      ;ENDFOLD
      ;FOLD -- ServoGun SZ1 oeffnen -- ;%{SE}%MKUKATPVW %CVW_COM %VCOMMENT %P 2:-- ServoGun SZ1 oeffnen --, 3: VW_COMMENT
      ;ENDFOLD
      ;FOLD A3511 = AUS ;%{SE}%MKUKATPVW %CVW_SPS %VBOASG %P 2:A3511 = AUS, 3: BOASG
         $OUT[3511] = FALSE
      ;ENDFOLD
      ;FOLD A3512 = EIN ;%{SE}%MKUKATPVW %CVW_SPS %VBOASG %P 2:A3512 = EIN, 3: BOASG
         $OUT[3512] = TRUE
      ;ENDFOLD
      ;FOLD -- RSK Fehlerausgabe Kraftaufbau -- ;%{SE}%MKUKATPVW %CVW_COM %VCOMMENT %P 2:-- RSK Fehlerausgabe Kraftaufbau --, 3: VW_COMMENT
      ;ENDFOLD
      ;FOLD F325 = AUS ;%{SE}%MKUKATPVW %CVW_SPS %VBOASG %P 2:F325 = AUS, 3: BOASG
         $FLAG[325] = FALSE
      ;ENDFOLD
      ;FOLD -- RSK Fehlerausgabe -- ;%{SE}%MKUKATPVW %CVW_COM %VCOMMENT %P 2:-- RSK Fehlerausgabe --, 3: VW_COMMENT
      ;ENDFOLD
      ;FOLD F327 = AUS ;%{SE}%MKUKATPVW %CVW_SPS %VBOASG %P 2:F327 = AUS, 3: BOASG
         $FLAG[327] = FALSE
      ;ENDFOLD
      ;FOLD -- RSK Fehlerausgabe -- ;%{SE}%MKUKATPVW %CVW_COM %VCOMMENT %P 2:-- RSK Fehlerausgabe --, 3: VW_COMMENT
      ;ENDFOLD
      ;FOLD F329 = AUS ;%{SE}%MKUKATPVW %CVW_SPS %VBOASG %P 2:F329 = AUS, 3: BOASG
         $FLAG[329] = FALSE
      ;ENDFOLD
      ;FOLD Schritt 234 = A3894 & A3506 & A3505 & !A3507 & A4039 ;%{SE}%MKUKATPVW %CVW_SPS %VST_CON %P 2:Schritt 234 = A3894 & A3506 & A3505 & !A3507 & A4039, 3: ST_CON
         IF $OUT[3894] AND $OUT[3506] AND $OUT[3505] AND NOT $OUT[3507] AND $OUT[4039] THEN
            PREV_STEP[9] = APP_INT_STEP[9]
            APP_INT_STEP[9] = 234
         ENDIF
      ;ENDFOLD
   ;ENDFOLD
   ;FOLD SCHRITT 234 -- st. RZ2 # Ende -- ;%{P}%MKUKATPVW,%CSTEP,%VST_NR,%P 1:SCHRITT, 2:234, 3: st. RZ2 # Ende
      ;FOLD ;%{H}
         Case 234
      ;ENDFOLD
      ;FOLD -- Hilfsflag SK Programmwechsel -- ;%{SE}%MKUKATPVW %CVW_COM %VCOMMENT %P 2:-- Hilfsflag SK Programmwechsel --, 3: VW_COMMENT
      ;ENDFOLD
      ;FOLD F334 = AUS ;%{SE}%MKUKATPVW %CVW_SPS %VBOASG %P 2:F334 = AUS, 3: BOASG
         $FLAG[334] = FALSE
      ;ENDFOLD
      ;FOLD A116 = AUS ;%{SE}%MKUKATPVW %CVW_SPS %VBOASG %P 2:A116 = AUS, 3: BOASG
         $OUT[116] = FALSE
      ;ENDFOLD
      ;FOLD A162 = AUS ;%{SE}%MKUKATPVW %CVW_SPS %VBOASG %P 2:A162 = AUS, 3: BOASG
         $OUT[162] = FALSE
      ;ENDFOLD
      ;FOLD A172 = AUS ;%{SE}%MKUKATPVW %CVW_SPS %VBOASG %P 2:A172 = AUS, 3: BOASG
         $OUT[172] = FALSE
      ;ENDFOLD
      ;FOLD A176 = AUS ;%{SE}%MKUKATPVW %CVW_SPS %VBOASG %P 2:A176 = AUS, 3: BOASG
         $OUT[176] = FALSE
      ;ENDFOLD
      ;FOLD A182 = AUS ;%{SE}%MKUKATPVW %CVW_SPS %VBOASG %P 2:A182 = AUS, 3: BOASG
         $OUT[182] = FALSE
      ;ENDFOLD
      ;FOLD A3518 = AUS ;%{SE}%MKUKATPVW %CVW_SPS %VBOASG %P 2:A3518 = AUS, 3: BOASG
         $OUT[3518] = FALSE
      ;ENDFOLD
      ;FOLD A3519 = AUS ;%{SE}%MKUKATPVW %CVW_SPS %VBOASG %P 2:A3519 = AUS, 3: BOASG
         $OUT[3519] = FALSE
      ;ENDFOLD
      ;FOLD A3533 = AUS ;%{SE}%MKUKATPVW %CVW_SPS %VBOASG %P 2:A3533 = AUS, 3: BOASG
         $OUT[3533] = FALSE
      ;ENDFOLD
      ;FOLD A947 = AUS ;%{SE}%MKUKATPVW %CVW_SPS %VBOASG %P 2:A947 = AUS, 3: BOASG
         $OUT[947] = FALSE
      ;ENDFOLD
      ;FOLD F748 = AUS ;%{SE}%MKUKATPVW %CVW_SPS %VBOASG %P 2:F748 = AUS, 3: BOASG
         $FLAG[748] = FALSE
      ;ENDFOLD
      ;FOLD F836 = AUS ;%{SE}%MKUKATPVW %CVW_SPS %VBOASG %P 2:F836 = AUS, 3: BOASG
         $FLAG[836] = FALSE
      ;ENDFOLD
      ;FOLD -- Start Init Same AUS -- ;%{SE}%MKUKATPVW %CVW_COM %VCOMMENT %P 2:-- Start Init Same AUS --, 3: VW_COMMENT
      ;ENDFOLD
      ;FOLD A3514 = AUS ;%{SE}%MKUKATPVW %CVW_SPS %VBOASG %P 2:A3514 = AUS, 3: BOASG
         $OUT[3514] = FALSE
      ;ENDFOLD
      ;FOLD -- Start Spot AUS -- ;%{SE}%MKUKATPVW %CVW_COM %VCOMMENT %P 2:-- Start Spot AUS --, 3: VW_COMMENT
      ;ENDFOLD
      ;FOLD A3511 = AUS ;%{SE}%MKUKATPVW %CVW_SPS %VBOASG %P 2:A3511 = AUS, 3: BOASG
         $OUT[3511] = FALSE
      ;ENDFOLD
      ;FOLD -- Start Dress AUS -- ;%{SE}%MKUKATPVW %CVW_COM %VCOMMENT %P 2:-- Start Dress AUS --, 3: VW_COMMENT
      ;ENDFOLD
      ;FOLD A3510 = AUS ;%{SE}%MKUKATPVW %CVW_SPS %VBOASG %P 2:A3510 = AUS, 3: BOASG
         $OUT[3510] = FALSE
      ;ENDFOLD
      ;FOLD -- Start Init New AUS -- ;%{SE}%MKUKATPVW %CVW_COM %VCOMMENT %P 2:-- Start Init New AUS --, 3: VW_COMMENT
      ;ENDFOLD
      ;FOLD A3513 = AUS ;%{SE}%MKUKATPVW %CVW_SPS %VBOASG %P 2:A3513 = AUS, 3: BOASG
         $OUT[3513] = FALSE
      ;ENDFOLD
      ;FOLD -- Dress in Position AUS -- ;%{SE}%MKUKATPVW %CVW_COM %VCOMMENT %P 2:-- Dress in Position AUS --, 3: VW_COMMENT
      ;ENDFOLD
      ;FOLD A3903 = AUS ;%{SE}%MKUKATPVW %CVW_SPS %VBOASG %P 2:A3903 = AUS, 3: BOASG
         $OUT[3903] = FALSE
      ;ENDFOLD
      ;FOLD -- Dress Fin AUS -- ;%{SE}%MKUKATPVW %CVW_COM %VCOMMENT %P 2:-- Dress Fin AUS --, 3: VW_COMMENT
      ;ENDFOLD
      ;FOLD A3904 = AUS ;%{SE}%MKUKATPVW %CVW_SPS %VBOASG %P 2:A3904 = AUS, 3: BOASG
         $OUT[3904] = FALSE
      ;ENDFOLD
      ;FOLD -- Start StartAcknowledge AUS -- ;%{SE}%MKUKATPVW %CVW_COM %VCOMMENT %P 2:-- Start StartAcknowledge AUS --, 3: VW_COMMENT
      ;ENDFOLD
      ;FOLD A3512 = AUS ;%{SE}%MKUKATPVW %CVW_SPS %VBOASG %P 2:A3512 = AUS, 3: BOASG
         $OUT[3512] = FALSE
      ;ENDFOLD
      ;FOLD -- RSK Sammelstoerung -- ;%{SE}%MKUKATPVW %CVW_COM %VCOMMENT %P 2:-- RSK Sammelstoerung --, 3: VW_COMMENT
      ;ENDFOLD
      ;FOLD F329 = F160 ;%{SE}%MKUKATPVW %CVW_SPS %VBOASG %P 2:F329 = F160, 3: BOASG
         $FLAG[329] = $FLAG[160]
      ;ENDFOLD
      ;FOLD F149 = (!E946 & E947 & !E948 & !F830) + F160 & (E26 + E27) ;%{SE}%MKUKATPVW %CVW_SPS %VBOASG %P 2:F149 = (!E946 & E947 & !E948 & !F830) + F160 & (E26 + E27), 3: BOASG
         $FLAG[149] = (NOT $IN[946] AND $IN[947] AND NOT $IN[948] AND NOT $FLAG[830]) OR $FLAG[160] AND ($IN[26] OR $IN[27])
      ;ENDFOLD
      ;FOLD Schritt 1 = F149 & A4039 & A3894 & A3506 & A3505 ;%{SE}%MKUKATPVW %CVW_SPS %VST_CON %P 2:Schritt 1 = F149 & A4039 & A3894 & A3506 & A3505, 3: ST_CON
         IF $FLAG[149] AND $OUT[4039] AND $OUT[3894] AND $OUT[3506] AND $OUT[3505] THEN
            PREV_STEP[9] = APP_INT_STEP[9]
            APP_INT_STEP[9] = 1
         ENDIF
      ;ENDFOLD
   ;ENDFOLD
   ;FOLD SCHRITT 250 -- st. RZ2 # Fehler Fraesen -- ;%{P}%MKUKATPVW,%CSTEP,%VST_NR,%P 1:SCHRITT, 2:250, 3: st. RZ2 # Fehler Fraesen
      ;FOLD ;%{H}
         Case 250
      ;ENDFOLD
      ;FOLD -- Ausblasen AUS -- ;%{SE}%MKUKATPVW %CVW_COM %VCOMMENT %P 2:-- Ausblasen AUS --, 3: VW_COMMENT
      ;ENDFOLD
      ;FOLD A996 = AUS ;%{SE}%MKUKATPVW %CVW_SPS %VBOASG %P 2:A996 = AUS, 3: BOASG
         $OUT[996] = FALSE
      ;ENDFOLD
      ;FOLD -- Fraesen AUS -- ;%{SE}%MKUKATPVW %CVW_COM %VCOMMENT %P 2:-- Fraesen AUS --, 3: VW_COMMENT
      ;ENDFOLD
      ;FOLD A994 = AUS ;%{SE}%MKUKATPVW %CVW_SPS %VBOASG %P 2:A994 = AUS, 3: BOASG
         $OUT[994] = FALSE
      ;ENDFOLD
      ;FOLD -- Fehler Reset EIN -- ;%{SE}%MKUKATPVW %CVW_COM %VCOMMENT %P 2:-- Fehler Reset EIN --, 3: VW_COMMENT
      ;ENDFOLD
      ;FOLD A3889 = EIN ;%{SE}%MKUKATPVW %CVW_SPS %VBOASG %P 2:A3889 = EIN, 3: BOASG
         $OUT[3889] = TRUE
      ;ENDFOLD
      ;FOLD -- Dress in Position AUS -- ;%{SE}%MKUKATPVW %CVW_COM %VCOMMENT %P 2:-- Dress in Position AUS --, 3: VW_COMMENT
      ;ENDFOLD
      ;FOLD A3903 = AUS ;%{SE}%MKUKATPVW %CVW_SPS %VBOASG %P 2:A3903 = AUS, 3: BOASG
         $OUT[3903] = FALSE
      ;ENDFOLD
      ;FOLD -- Start Dress Fin AUS -- ;%{SE}%MKUKATPVW %CVW_COM %VCOMMENT %P 2:-- Start Dress Fin AUS --, 3: VW_COMMENT
      ;ENDFOLD
      ;FOLD A3904 = AUS ;%{SE}%MKUKATPVW %CVW_SPS %VBOASG %P 2:A3904 = AUS, 3: BOASG
         $OUT[3904] = FALSE
      ;ENDFOLD
      ;FOLD -- Fehler An SPS EIN -- ;%{SE}%MKUKATPVW %CVW_COM %VCOMMENT %P 2:-- Fehler An SPS EIN --, 3: VW_COMMENT
      ;ENDFOLD
      ;FOLD A172 = EIN ;%{SE}%MKUKATPVW %CVW_SPS %VBOASG %P 2:A172 = EIN, 3: BOASG
         $OUT[172] = TRUE
      ;ENDFOLD
      ;FOLD -- Anwahl Zange 1 EIN -- ;%{SE}%MKUKATPVW %CVW_COM %VCOMMENT %P 2:-- Anwahl Zange 1 EIN --, 3: VW_COMMENT
      ;ENDFOLD
      ;FOLD A3890 = EIN ;%{SE}%MKUKATPVW %CVW_SPS %VBOASG %P 2:A3890 = EIN, 3: BOASG
         $OUT[3890] = TRUE
      ;ENDFOLD
      ;FOLD -- Ueberwachungszeit Fehler Fraesen -- ;%{SE}%MKUKATPVW %CVW_COM %VCOMMENT %P 2:-- Ueberwachungszeit Fehler Fraesen --, 3: VW_COMMENT
      ;ENDFOLD
      ;FOLD t11 ( EIN ) = STOP ;%{SE}%MKUKATPVW %CVW_SPS %VTSTOP %P 2:t11 ( EIN ) = STOP, 3: TSTOP
         VW(#SET_TIME,TRUE,11,1,0)
      ;ENDFOLD
      ;FOLD F328 = AUS ;%{SE}%MKUKATPVW %CVW_SPS %VBOASG %P 2:F328 = AUS, 3: BOASG
         $FLAG[328] = FALSE
      ;ENDFOLD
      ;FOLD F324 = AUS ;%{SE}%MKUKATPVW %CVW_SPS %VBOASG %P 2:F324 = AUS, 3: BOASG
         $FLAG[324] = FALSE
      ;ENDFOLD
      ;FOLD Schritt 251 = A4039 ;%{SE}%MKUKATPVW %CVW_SPS %VST_CON %P 2:Schritt 251 = A4039, 3: ST_CON
         IF $OUT[4039] THEN
            PREV_STEP[9] = APP_INT_STEP[9]
            APP_INT_STEP[9] = 251
         ENDIF
      ;ENDFOLD
   ;ENDFOLD
   ;FOLD SCHRITT 251 -- st. RZ2 # Fehler Fraesen -- ;%{P}%MKUKATPVW,%CSTEP,%VST_NR,%P 1:SCHRITT, 2:251, 3: st. RZ2 # Fehler Fraesen
      ;FOLD ;%{H}
         Case 251
      ;ENDFOLD
      ;FOLD -- Fehler Reset AUS -- ;%{SE}%MKUKATPVW %CVW_COM %VCOMMENT %P 2:-- Fehler Reset AUS --, 3: VW_COMMENT
      ;ENDFOLD
      ;FOLD A3889 = AUS ;%{SE}%MKUKATPVW %CVW_SPS %VBOASG %P 2:A3889 = AUS, 3: BOASG
         $OUT[3889] = FALSE
      ;ENDFOLD
      ;FOLD -- Start StartAcknowledge EIN -- ;%{SE}%MKUKATPVW %CVW_COM %VCOMMENT %P 2:-- Start StartAcknowledge EIN --, 3: VW_COMMENT
      ;ENDFOLD
      ;FOLD A3512 = EIN ;%{SE}%MKUKATPVW %CVW_SPS %VBOASG %P 2:A3512 = EIN, 3: BOASG
         $OUT[3512] = TRUE
      ;ENDFOLD
      ;FOLD Schritt 252 = A4039 ;%{SE}%MKUKATPVW %CVW_SPS %VST_CON %P 2:Schritt 252 = A4039, 3: ST_CON
         IF $OUT[4039] THEN
            PREV_STEP[9] = APP_INT_STEP[9]
            APP_INT_STEP[9] = 252
         ENDIF
      ;ENDFOLD
   ;ENDFOLD
   ;FOLD SCHRITT 252 -- st. RZ2 # Fehler Fraesen -- ;%{P}%MKUKATPVW,%CSTEP,%VST_NR,%P 1:SCHRITT, 2:252, 3: st. RZ2 # Fehler Fraesen
      ;FOLD ;%{H}
         Case 252
      ;ENDFOLD
      ;FOLD -- Start StartAcknowledge AUS -- ;%{SE}%MKUKATPVW %CVW_COM %VCOMMENT %P 2:-- Start StartAcknowledge AUS --, 3: VW_COMMENT
      ;ENDFOLD
      ;FOLD A3512 = AUS ;%{SE}%MKUKATPVW %CVW_SPS %VBOASG %P 2:A3512 = AUS, 3: BOASG
         $OUT[3512] = FALSE
      ;ENDFOLD
      ;FOLD -- Start Dress in Position AUS -- ;%{SE}%MKUKATPVW %CVW_COM %VCOMMENT %P 2:-- Start Dress in Position AUS --, 3: VW_COMMENT
      ;ENDFOLD
      ;FOLD A3903 = AUS ;%{SE}%MKUKATPVW %CVW_SPS %VBOASG %P 2:A3903 = AUS, 3: BOASG
         $OUT[3903] = FALSE
      ;ENDFOLD
      ;FOLD -- Start Dress Fin AUS -- ;%{SE}%MKUKATPVW %CVW_COM %VCOMMENT %P 2:-- Start Dress Fin AUS --, 3: VW_COMMENT
      ;ENDFOLD
      ;FOLD A3904 = AUS ;%{SE}%MKUKATPVW %CVW_SPS %VBOASG %P 2:A3904 = AUS, 3: BOASG
         $OUT[3904] = FALSE
      ;ENDFOLD
      ;FOLD -- Start Dress AUS -- ;%{SE}%MKUKATPVW %CVW_COM %VCOMMENT %P 2:-- Start Dress AUS --, 3: VW_COMMENT
      ;ENDFOLD
      ;FOLD A3510 = EIN ;%{SE}%MKUKATPVW %CVW_SPS %VBOASG %P 2:A3510 = EIN, 3: BOASG
         $OUT[3510] = TRUE
      ;ENDFOLD
      ;FOLD -- Start Spot AUS -- ;%{SE}%MKUKATPVW %CVW_COM %VCOMMENT %P 2:-- Start Spot AUS --, 3: VW_COMMENT
      ;ENDFOLD
      ;FOLD A3511 = AUS ;%{SE}%MKUKATPVW %CVW_SPS %VBOASG %P 2:A3511 = AUS, 3: BOASG
         $OUT[3511] = FALSE
      ;ENDFOLD
      ;FOLD -- Start Spot AUS -- ;%{SE}%MKUKATPVW %CVW_COM %VCOMMENT %P 2:-- Start Spot AUS --, 3: VW_COMMENT
      ;ENDFOLD
      ;FOLD A3511 = AUS ;%{SE}%MKUKATPVW %CVW_SPS %VBOASG %P 2:A3511 = AUS, 3: BOASG
         $OUT[3511] = FALSE
      ;ENDFOLD
      ;FOLD -- Start Init Same AUS -- ;%{SE}%MKUKATPVW %CVW_COM %VCOMMENT %P 2:-- Start Init Same AUS --, 3: VW_COMMENT
      ;ENDFOLD
      ;FOLD A3514 = AUS ;%{SE}%MKUKATPVW %CVW_SPS %VBOASG %P 2:A3514 = AUS, 3: BOASG
         $OUT[3514] = FALSE
      ;ENDFOLD
      ;FOLD -- Start Init New AUS -- ;%{SE}%MKUKATPVW %CVW_COM %VCOMMENT %P 2:-- Start Init New AUS --, 3: VW_COMMENT
      ;ENDFOLD
      ;FOLD A3513 = AUS ;%{SE}%MKUKATPVW %CVW_SPS %VBOASG %P 2:A3513 = AUS, 3: BOASG
         $OUT[3513] = FALSE
      ;ENDFOLD
      ;FOLD A3518 = A3519 ;%{SE}%MKUKATPVW %CVW_SPS %VBOASG %P 2:A3518 = A3519, 3: BOASG
         $OUT[3518] = $OUT[3519]
      ;ENDFOLD
      ;FOLD Schritt 253 = A4039 & A3864 ;%{SE}%MKUKATPVW %CVW_SPS %VST_CON %P 2:Schritt 253 = A4039 & A3864, 3: ST_CON
         IF $OUT[4039] AND $OUT[3864] THEN
            PREV_STEP[9] = APP_INT_STEP[9]
            APP_INT_STEP[9] = 253
         ENDIF
      ;ENDFOLD
   ;ENDFOLD
   ;FOLD SCHRITT 253 -- st. RZ2 # Fehler Fraesen -- ;%{P}%MKUKATPVW,%CSTEP,%VST_NR,%P 1:SCHRITT, 2:253, 3: st. RZ2 # Fehler Fraesen
      ;FOLD ;%{H}
         Case 253
      ;ENDFOLD
      ;FOLD -- RSK Fehlerausgabe KF Versetzeinheit -- ;%{SE}%MKUKATPVW %CVW_COM %VCOMMENT %P 2:-- RSK Fehlerausgabe KF Versetzeinheit --, 3: VW_COMMENT
      ;ENDFOLD
      ;FOLD F328 = E995 & F564 ;%{SE}%MKUKATPVW %CVW_SPS %VBOASG %P 2:F328 = E995 & F564, 3: BOASG
         $FLAG[328] = $IN[995] AND $FLAG[564]
      ;ENDFOLD
      ;FOLD -- RSK Fehlerausgabe KS1 Arbeitsstellung -- ;%{SE}%MKUKATPVW %CVW_COM %VCOMMENT %P 2:-- RSK Fehlerausgabe KS1 Arbeitsstellung --, 3: VW_COMMENT
      ;ENDFOLD
      ;FOLD F324 = (E996 + !E997 + !E998 + E999) ;%{SE}%MKUKATPVW %CVW_SPS %VBOASG %P 2:F324 = (E996 + !E997 + !E998 + E999), 3: BOASG
         $FLAG[324] = ($IN[996] OR NOT $IN[997] OR NOT $IN[998] OR $IN[999])
      ;ENDFOLD
      ;FOLD A3519 = EIN ;%{SE}%MKUKATPVW %CVW_SPS %VBOASG %P 2:A3519 = EIN, 3: BOASG
         $OUT[3519] = TRUE
      ;ENDFOLD
      ;FOLD Schritt 254 = A4039 & A3894 & A3505 & A3506 & !A3518 & (E26 + E27) ;%{SE}%MKUKATPVW %CVW_SPS %VST_CON %P 2:Schritt 254 = A4039 & A3894 & A3505 & A3506 & !A3518 & (E26 + E27), 3: ST_CON
         IF $OUT[4039] AND $OUT[3894] AND $OUT[3505] AND $OUT[3506] AND NOT $OUT[3518] AND ($IN[26] OR $IN[27]) THEN
            PREV_STEP[9] = APP_INT_STEP[9]
            APP_INT_STEP[9] = 254
         ENDIF
      ;ENDFOLD
      ;FOLD Schritt 216 = A4039 & A3894 & A3505 & A3506 & A3518 & (E26 + E27) ;%{SE}%MKUKATPVW %CVW_SPS %VST_CON %P 2:Schritt 216 = A4039 & A3894 & A3505 & A3506 & A3518 & (E26 + E27), 3: ST_CON
         IF $OUT[4039] AND $OUT[3894] AND $OUT[3505] AND $OUT[3506] AND $OUT[3518] AND ($IN[26] OR $IN[27]) THEN
            PREV_STEP[9] = APP_INT_STEP[9]
            APP_INT_STEP[9] = 216
         ENDIF
      ;ENDFOLD
   ;ENDFOLD
   ;FOLD SCHRITT 254 -- st. RZ2 # Fehler Fraesen -- ;%{P}%MKUKATPVW,%CSTEP,%VST_NR,%P 1:SCHRITT, 2:254, 3: st. RZ2 # Fehler Fraesen
      ;FOLD ;%{H}
         Case 254
      ;ENDFOLD
      ;FOLD -- Fehler ruecksetzen -- ;%{SE}%MKUKATPVW %CVW_COM %VCOMMENT %P 2:-- Fehler ruecksetzen --, 3: VW_COMMENT
      ;ENDFOLD
      ;FOLD A172 = AUS ;%{SE}%MKUKATPVW %CVW_SPS %VBOASG %P 2:A172 = AUS, 3: BOASG
         $OUT[172] = FALSE
      ;ENDFOLD
      ;FOLD A176 = AUS ;%{SE}%MKUKATPVW %CVW_SPS %VBOASG %P 2:A176 = AUS, 3: BOASG
         $OUT[176] = FALSE
      ;ENDFOLD
      ;FOLD Schritt 203 = (F324 + F328) & E996 & !E997 & !E998 & E999 & A4039 ;%{SE}%MKUKATPVW %CVW_SPS %VST_CON %P 2:Schritt 203 = (F324 + F328) & E996 & !E997 & !E998 & E999 & A4039, 3: ST_CON
         IF ($FLAG[324] OR $FLAG[328]) AND $IN[996] AND NOT $IN[997] AND NOT $IN[998] AND $IN[999] AND $OUT[4039] THEN
            PREV_STEP[9] = APP_INT_STEP[9]
            APP_INT_STEP[9] = 203
         ENDIF
      ;ENDFOLD
      ;FOLD SCHRITT 211 = !F324 & !F328 & !E996 & E997 & E998 & !E999 & A4039 ;%{SE}%MKUKATPVW %CVW_SPS %VST_CON %P 2:SCHRITT 211 = !F324 & !F328 & !E996 & E997 & E998 & !E999 & A4039, 3: ST_CON
         IF NOT $FLAG[324] AND NOT $FLAG[328] AND NOT $IN[996] AND $IN[997] AND $IN[998] AND NOT $IN[999] AND $OUT[4039] THEN
            PREV_STEP[9] = APP_INT_STEP[9]
            APP_INT_STEP[9] = 211
         ENDIF
      ;ENDFOLD
   ;ENDFOLD
   ;FOLD SCHRITT 255 -- st. RZ2 # Fehler Fraesen  -- ;%{P}%MKUKATPVW,%CSTEP,%VST_NR,%P 1:SCHRITT, 2:255, 3: st. RZ2 # Fehler Fraesen
      ;FOLD ;%{H}
         Case 255
      ;ENDFOLD
      ;FOLD Schritt 211 = A4039 & A3506 & A3505 ;%{SE}%MKUKATPVW %CVW_SPS %VST_CON %P 2:Schritt 211 = A4039 & A3506 & A3505, 3: ST_CON
         IF $OUT[4039] AND $OUT[3506] AND $OUT[3505] THEN
            PREV_STEP[9] = APP_INT_STEP[9]
            APP_INT_STEP[9] = 211
         ENDIF
      ;ENDFOLD
   ;ENDFOLD
   ;FOLD SCHRITT 260 -- st. RZ2 # Fehler Messen -- ;%{P}%MKUKATPVW,%CSTEP,%VST_NR,%P 1:SCHRITT, 2:260, 3: st. RZ2 # Fehler Messen
      ;FOLD ;%{H}
         Case 260
      ;ENDFOLD
      ;FOLD 1:;%{SE} %MKUKATPVW
      ;ENDFOLD
   ;ENDFOLD
   ;FOLD SCHRITT 261 -- st. RZ2 # Fehler Messen -- ;%{P}%MKUKATPVW,%CSTEP,%VST_NR,%P 1:SCHRITT, 2:261, 3: st. RZ2 # Fehler Messen
      ;FOLD ;%{H}
         Case 261
      ;ENDFOLD
      ;FOLD -- Fehler Reset AUS -- ;%{SE}%MKUKATPVW %CVW_COM %VCOMMENT %P 2:-- Fehler Reset AUS --, 3: VW_COMMENT
      ;ENDFOLD
      ;FOLD A3889 = AUS ;%{SE}%MKUKATPVW %CVW_SPS %VBOASG %P 2:A3889 = AUS, 3: BOASG
         $OUT[3889] = FALSE
      ;ENDFOLD
      ;FOLD -- Anwahl Zange 1 EIN -- ;%{SE}%MKUKATPVW %CVW_COM %VCOMMENT %P 2:-- Anwahl Zange 1 EIN --, 3: VW_COMMENT
      ;ENDFOLD
      ;FOLD A3890 = EIN ;%{SE}%MKUKATPVW %CVW_SPS %VBOASG %P 2:A3890 = EIN, 3: BOASG
         $OUT[3890] = TRUE
      ;ENDFOLD
      ;FOLD -- Start StartAcknowledge EIN -- ;%{SE}%MKUKATPVW %CVW_COM %VCOMMENT %P 2:-- Start StartAcknowledge EIN --, 3: VW_COMMENT
      ;ENDFOLD
      ;FOLD A3512 = EIN ;%{SE}%MKUKATPVW %CVW_SPS %VBOASG %P 2:A3512 = EIN, 3: BOASG
         $OUT[3512] = TRUE
      ;ENDFOLD
      ;FOLD Schritt 262 = A4039 & A172 & A3894 ;%{SE}%MKUKATPVW %CVW_SPS %VST_CON %P 2:Schritt 262 = A4039 & A172 & A3894, 3: ST_CON
         IF $OUT[4039] AND $OUT[172] AND $OUT[3894] THEN
            PREV_STEP[9] = APP_INT_STEP[9]
            APP_INT_STEP[9] = 262
         ENDIF
      ;ENDFOLD
   ;ENDFOLD
   ;FOLD SCHRITT 262 -- st. RZ2 # Fehler Messen -- ;%{P}%MKUKATPVW,%CSTEP,%VST_NR,%P 1:SCHRITT, 2:262, 3: st. RZ2 # Fehler Messen
      ;FOLD ;%{H}
         Case 262
      ;ENDFOLD
      ;FOLD -- Start Init Same AUS -- ;%{SE}%MKUKATPVW %CVW_COM %VCOMMENT %P 2:-- Start Init Same AUS --, 3: VW_COMMENT
      ;ENDFOLD
      ;FOLD A3514 = AUS ;%{SE}%MKUKATPVW %CVW_SPS %VBOASG %P 2:A3514 = AUS, 3: BOASG
         $OUT[3514] = FALSE
      ;ENDFOLD
      ;FOLD -- Start Spot AUS -- ;%{SE}%MKUKATPVW %CVW_COM %VCOMMENT %P 2:-- Start Spot AUS --, 3: VW_COMMENT
      ;ENDFOLD
      ;FOLD A3511 = AUS ;%{SE}%MKUKATPVW %CVW_SPS %VBOASG %P 2:A3511 = AUS, 3: BOASG
         $OUT[3511] = FALSE
      ;ENDFOLD
      ;FOLD -- Start Dress AUS -- ;%{SE}%MKUKATPVW %CVW_COM %VCOMMENT %P 2:-- Start Dress AUS --, 3: VW_COMMENT
      ;ENDFOLD
      ;FOLD A3510 = AUS ;%{SE}%MKUKATPVW %CVW_SPS %VBOASG %P 2:A3510 = AUS, 3: BOASG
         $OUT[3510] = FALSE
      ;ENDFOLD
      ;FOLD -- Start Init New AUS -- ;%{SE}%MKUKATPVW %CVW_COM %VCOMMENT %P 2:-- Start Init New AUS --, 3: VW_COMMENT
      ;ENDFOLD
      ;FOLD A3513 = AUS ;%{SE}%MKUKATPVW %CVW_SPS %VBOASG %P 2:A3513 = AUS, 3: BOASG
         $OUT[3513] = FALSE
      ;ENDFOLD
      ;FOLD -- Start Dress in Position AUS -- ;%{SE}%MKUKATPVW %CVW_COM %VCOMMENT %P 2:-- Start Dress in Position AUS --, 3: VW_COMMENT
      ;ENDFOLD
      ;FOLD A3903 = AUS ;%{SE}%MKUKATPVW %CVW_SPS %VBOASG %P 2:A3903 = AUS, 3: BOASG
         $OUT[3903] = FALSE
      ;ENDFOLD
      ;FOLD -- Start Dress Fin AUS -- ;%{SE}%MKUKATPVW %CVW_COM %VCOMMENT %P 2:-- Start Dress Fin AUS --, 3: VW_COMMENT
      ;ENDFOLD
      ;FOLD A3904 = AUS ;%{SE}%MKUKATPVW %CVW_SPS %VBOASG %P 2:A3904 = AUS, 3: BOASG
         $OUT[3904] = FALSE
      ;ENDFOLD
      ;FOLD -- Start StartAcknowledge AUS -- ;%{SE}%MKUKATPVW %CVW_COM %VCOMMENT %P 2:-- Start StartAcknowledge AUS --, 3: VW_COMMENT
      ;ENDFOLD
      ;FOLD A3512 = AUS ;%{SE}%MKUKATPVW %CVW_SPS %VBOASG %P 2:A3512 = AUS, 3: BOASG
         $OUT[3512] = FALSE
      ;ENDFOLD
      ;FOLD Schritt 263 = A4039 ;%{SE}%MKUKATPVW %CVW_SPS %VST_CON %P 2:Schritt 263 = A4039, 3: ST_CON
         IF $OUT[4039] THEN
            PREV_STEP[9] = APP_INT_STEP[9]
            APP_INT_STEP[9] = 263
         ENDIF
      ;ENDFOLD
   ;ENDFOLD
   ;FOLD SCHRITT 263 -- st. RZ2 # Fehler Messen -- ;%{P}%MKUKATPVW,%CSTEP,%VST_NR,%P 1:SCHRITT, 2:263, 3: st. RZ2 # Fehler Messen
      ;FOLD ;%{H}
         Case 263
      ;ENDFOLD
      ;FOLD Schritt 264 = A4039 & !A3507 & A3506 & (E26 + E27) ;%{SE}%MKUKATPVW %CVW_SPS %VST_CON %P 2:Schritt 264 = A4039 & !A3507 & A3506 & (E26 + E27), 3: ST_CON
         IF $OUT[4039] AND NOT $OUT[3507] AND $OUT[3506] AND ($IN[26] OR $IN[27]) THEN
            PREV_STEP[9] = APP_INT_STEP[9]
            APP_INT_STEP[9] = 264
         ENDIF
      ;ENDFOLD
   ;ENDFOLD
   ;FOLD SCHRITT 264 -- st. RZ2 # Fehler Messen -- ;%{P}%MKUKATPVW,%CSTEP,%VST_NR,%P 1:SCHRITT, 2:264, 3: st. RZ2 # Fehler Messen
      ;FOLD ;%{H}
         Case 264
      ;ENDFOLD
      ;FOLD Schritt 224 = A4039 & A172 & !A3507 & A3506 & A3505 ;%{SE}%MKUKATPVW %CVW_SPS %VST_CON %P 2:Schritt 224 = A4039 & A172 & !A3507 & A3506 & A3505, 3: ST_CON
         IF $OUT[4039] AND $OUT[172] AND NOT $OUT[3507] AND $OUT[3506] AND $OUT[3505] THEN
            PREV_STEP[9] = APP_INT_STEP[9]
            APP_INT_STEP[9] = 224
         ENDIF
      ;ENDFOLD
   ;ENDFOLD
   ;FOLD SCHRITT 265 -- st. RZ2 # Fehler Schweissen-- ;%{P}%MKUKATPVW,%CSTEP,%VST_NR,%P 1:SCHRITT, 2:265, 3: st. RZ2 # Fehler Schweissen
      ;FOLD ;%{H}
         Case 265
      ;ENDFOLD
      ;FOLD -- Start StartAcknowledge AUS -- ;%{SE}%MKUKATPVW %CVW_COM %VCOMMENT %P 2:-- Start StartAcknowledge AUS --, 3: VW_COMMENT
      ;ENDFOLD
      ;FOLD A3512 = AUS ;%{SE}%MKUKATPVW %CVW_SPS %VBOASG %P 2:A3512 = AUS, 3: BOASG
         $OUT[3512] = FALSE
      ;ENDFOLD
      ;FOLD -- Start Dress in Position AUS -- ;%{SE}%MKUKATPVW %CVW_COM %VCOMMENT %P 2:-- Start Dress in Position AUS --, 3: VW_COMMENT
      ;ENDFOLD
      ;FOLD A3903 = AUS ;%{SE}%MKUKATPVW %CVW_SPS %VBOASG %P 2:A3903 = AUS, 3: BOASG
         $OUT[3903] = FALSE
      ;ENDFOLD
      ;FOLD -- Start Dress Fin AUS -- ;%{SE}%MKUKATPVW %CVW_COM %VCOMMENT %P 2:-- Start Dress Fin AUS --, 3: VW_COMMENT
      ;ENDFOLD
      ;FOLD A3904 = AUS ;%{SE}%MKUKATPVW %CVW_SPS %VBOASG %P 2:A3904 = AUS, 3: BOASG
         $OUT[3904] = FALSE
      ;ENDFOLD
      ;FOLD -- Start Dress AUS -- ;%{SE}%MKUKATPVW %CVW_COM %VCOMMENT %P 2:-- Start Dress AUS --, 3: VW_COMMENT
      ;ENDFOLD
      ;FOLD A3510 = AUS ;%{SE}%MKUKATPVW %CVW_SPS %VBOASG %P 2:A3510 = AUS, 3: BOASG
         $OUT[3510] = FALSE
      ;ENDFOLD
      ;FOLD -- Start Spot AUS -- ;%{SE}%MKUKATPVW %CVW_COM %VCOMMENT %P 2:-- Start Spot AUS --, 3: VW_COMMENT
      ;ENDFOLD
      ;FOLD A3511 = AUS ;%{SE}%MKUKATPVW %CVW_SPS %VBOASG %P 2:A3511 = AUS, 3: BOASG
         $OUT[3511] = FALSE
      ;ENDFOLD
      ;FOLD -- Start Spot AUS -- ;%{SE}%MKUKATPVW %CVW_COM %VCOMMENT %P 2:-- Start Spot AUS --, 3: VW_COMMENT
      ;ENDFOLD
      ;FOLD A3511 = AUS ;%{SE}%MKUKATPVW %CVW_SPS %VBOASG %P 2:A3511 = AUS, 3: BOASG
         $OUT[3511] = FALSE
      ;ENDFOLD
      ;FOLD -- Start Init Same AUS -- ;%{SE}%MKUKATPVW %CVW_COM %VCOMMENT %P 2:-- Start Init Same AUS --, 3: VW_COMMENT
      ;ENDFOLD
      ;FOLD A3514 = AUS ;%{SE}%MKUKATPVW %CVW_SPS %VBOASG %P 2:A3514 = AUS, 3: BOASG
         $OUT[3514] = FALSE
      ;ENDFOLD
      ;FOLD -- Start Init New AUS -- ;%{SE}%MKUKATPVW %CVW_COM %VCOMMENT %P 2:-- Start Init New AUS --, 3: VW_COMMENT
      ;ENDFOLD
      ;FOLD A3513 = AUS ;%{SE}%MKUKATPVW %CVW_SPS %VBOASG %P 2:A3513 = AUS, 3: BOASG
         $OUT[3513] = FALSE
      ;ENDFOLD
      ;FOLD A3533 = EIN ;%{SE}%MKUKATPVW %CVW_SPS %VBOASG %P 2:A3533 = EIN, 3: BOASG
         $OUT[3533] = TRUE
      ;ENDFOLD
      ;FOLD A162 = AUS ;%{SE}%MKUKATPVW %CVW_SPS %VBOASG %P 2:A162 = AUS, 3: BOASG
         $OUT[162] = FALSE
      ;ENDFOLD
      ;FOLD F148 = AUS ;%{SE}%MKUKATPVW %CVW_SPS %VBOASG %P 2:F148 = AUS, 3: BOASG
         $FLAG[148] = FALSE
      ;ENDFOLD
      ;FOLD Schritt 2 = A4039 & A3894 & A3506 & A3505 & (E26 + E27) ;%{SE}%MKUKATPVW %CVW_SPS %VST_CON %P 2:Schritt 2 = A4039 & A3894 & A3506 & A3505 & (E26 + E27), 3: ST_CON
         IF $OUT[4039] AND $OUT[3894] AND $OUT[3506] AND $OUT[3505] AND ($IN[26] OR $IN[27]) THEN
            PREV_STEP[9] = APP_INT_STEP[9]
            APP_INT_STEP[9] = 2
         ENDIF
      ;ENDFOLD
   ;ENDFOLD
   ;FOLD SCHRITT 266 -- st. RZ2 # Fehler Schweissen-- ;%{P}%MKUKATPVW,%CSTEP,%VST_NR,%P 1:SCHRITT, 2:266, 3: st. RZ2 # Fehler Schweissen
      ;FOLD ;%{H}
         Case 266
      ;ENDFOLD
      ;FOLD 1:;%{SE} %MKUKATPVW
      ;ENDFOLD
   ;ENDFOLD
   ;FOLD SCHRITT 290 -- st. RZ2 Setzhub 2 -- ;%{P}%MKUKATPVW,%CSTEP,%VST_NR,%P 1:SCHRITT, 2:290, 3: st. RZ2 Setzhub 2
      ;FOLD ;%{H}
         Case 290
      ;ENDFOLD
      ;FOLD -- Druckvorgabe SK1/ServoGun -- ;%{SE}%MKUKATPVW %CVW_COM %VCOMMENT %P 2:-- Druckvorgabe SK1/ServoGun --, 3: VW_COMMENT
      ;ENDFOLD
      ;FOLD bin4 ( F138 ) = 61 ;%{SE}%MKUKATPVW %CVW_SPS %VARIASG %P 2:bin4 ( F138 ) = 61, 3: ARIASG
         VW(#BINOUT,$FLAG[138],4,61)
      ;ENDFOLD
      ;FOLD bin31 ( F138 ) = 61 ;%{SE}%MKUKATPVW %CVW_SPS %VARIASG %P 2:bin31 ( F138 ) = 61, 3: ARIASG
         VW(#BINOUT,$FLAG[138],31,61)
      ;ENDFOLD
      ;FOLD -- Wartezeit Programmwechsel SK -- ;%{SE}%MKUKATPVW %CVW_COM %VCOMMENT %P 2:-- Wartezeit Programmwechsel SK --, 3: VW_COMMENT
      ;ENDFOLD
      ;FOLD T8 ( !F334 ) = -2[1/10Sek] ;%{SE}%MKUKATPVW %CVW_SPS %VTASG %P 2:T8 ( !F334 ) = -2[1/10Sek], 3: TASG
         VW(#SET_TIME,NOT $FLAG[334],8,0,-2)
      ;ENDFOLD
      ;FOLD -- Ueberwachungszeit ServoGun Setzhub 2 -- ;%{SE}%MKUKATPVW %CVW_COM %VCOMMENT %P 2:-- Ueberwachungszeit ServoGun Setzhub 2 --, 3: VW_COMMENT
      ;ENDFOLD
      ;FOLD t9 ( EIN ) = -80[1/10Sek] ;%{SE}%MKUKATPVW %CVW_SPS %VTASG %P 2:t9 ( EIN ) = -80[1/10Sek], 3: TASG
         VW(#SET_TIME,TRUE,9,0,-80)
      ;ENDFOLD
      ;FOLD -- Hilfsflag SK Programmwechsel -- ;%{SE}%MKUKATPVW %CVW_COM %VCOMMENT %P 2:-- Hilfsflag SK Programmwechsel --, 3: VW_COMMENT
      ;ENDFOLD
      ;FOLD F334 = EIN ;%{SE}%MKUKATPVW %CVW_SPS %VBOASG %P 2:F334 = EIN, 3: BOASG
         $FLAG[334] = TRUE
      ;ENDFOLD
      ;FOLD A3512 = AUS ;%{SE}%MKUKATPVW %CVW_SPS %VBOASG %P 2:A3512 = AUS, 3: BOASG
         $OUT[3512] = FALSE
      ;ENDFOLD
      ;FOLD SCHRITT 291 = T8 & A4039 & A3506 & A3505 & !A3507 ;%{SE}%MKUKATPVW %CVW_SPS %VST_CON %P 2:SCHRITT 291 = T8 & A4039 & A3506 & A3505 & !A3507, 3: ST_CON
         IF $TIMER_FLAG[8] AND $OUT[4039] AND $OUT[3506] AND $OUT[3505] AND NOT $OUT[3507] THEN
            PREV_STEP[9] = APP_INT_STEP[9]
            APP_INT_STEP[9] = 291
         ENDIF
      ;ENDFOLD
   ;ENDFOLD
   ;FOLD SCHRITT 291 -- st. RZ2 Setzhub 2 # InitSame -- ;%{P}%MKUKATPVW,%CSTEP,%VST_NR,%P 1:SCHRITT, 2:291, 3: st. RZ2 Setzhub 2 # InitSame
      ;FOLD ;%{H}
         Case 291
      ;ENDFOLD
      ;FOLD -- Hilfsflag SK Programmwechsel -- ;%{SE}%MKUKATPVW %CVW_COM %VCOMMENT %P 2:-- Hilfsflag SK Programmwechsel --, 3: VW_COMMENT
      ;ENDFOLD
      ;FOLD F334 = AUS ;%{SE}%MKUKATPVW %CVW_SPS %VBOASG %P 2:F334 = AUS, 3: BOASG
         $FLAG[334] = FALSE
      ;ENDFOLD
      ;FOLD -- Zeit fuer Setzhub -- ;%{SE}%MKUKATPVW %CVW_COM %VCOMMENT %P 2:-- Zeit fuer Setzhub --, 3: VW_COMMENT
      ;ENDFOLD
      ;FOLD T8 ( EIN ) = -80[1/10Sek] ;%{SE}%MKUKATPVW %CVW_SPS %VTASG %P 2:T8 ( EIN ) = -80[1/10Sek], 3: TASG
         VW(#SET_TIME,TRUE,8,0,-80)
      ;ENDFOLD
      ;FOLD -- Messen nach Fraesen -- ;%{SE}%MKUKATPVW %CVW_COM %VCOMMENT %P 2:-- Messen nach Fraesen --, 3: VW_COMMENT
      ;ENDFOLD
      ;FOLD A3514 = EIN ;%{SE}%MKUKATPVW %CVW_SPS %VBOASG %P 2:A3514 = EIN, 3: BOASG
         $OUT[3514] = TRUE
      ;ENDFOLD
      ;FOLD A3510 = EIN ;%{SE}%MKUKATPVW %CVW_SPS %VBOASG %P 2:A3510 = EIN, 3: BOASG
         $OUT[3510] = TRUE
      ;ENDFOLD
      ;FOLD SCHRITT 292 = A4039 ;%{SE}%MKUKATPVW %CVW_SPS %VST_CON %P 2:SCHRITT 292 = A4039, 3: ST_CON
         IF $OUT[4039] THEN
            PREV_STEP[9] = APP_INT_STEP[9]
            APP_INT_STEP[9] = 292
         ENDIF
      ;ENDFOLD
   ;ENDFOLD
   ;FOLD SCHRITT 292 -- st. RZ2 Setzhub 2 # Auswertung -- ;%{P}%MKUKATPVW,%CSTEP,%VST_NR,%P 1:SCHRITT, 2:292, 3: st. RZ2 Setzhub 2 # Auswertung
      ;FOLD ;%{H}
         Case 292
      ;ENDFOLD
      ;FOLD -- Hilfsflag SK Programmwechsel -- ;%{SE}%MKUKATPVW %CVW_COM %VCOMMENT %P 2:-- Hilfsflag SK Programmwechsel --, 3: VW_COMMENT
      ;ENDFOLD
      ;FOLD F334 = AUS ;%{SE}%MKUKATPVW %CVW_SPS %VBOASG %P 2:F334 = AUS, 3: BOASG
         $FLAG[334] = FALSE
      ;ENDFOLD
      ;FOLD -- Warte Ergebnis -- ;%{SE}%MKUKATPVW %CVW_COM %VCOMMENT %P 2:-- Warte Ergebnis --, 3: VW_COMMENT
      ;ENDFOLD
      ;FOLD SCHRITT 293 = A3508 & A4039 + T8 + T9 ;%{SE}%MKUKATPVW %CVW_SPS %VST_CON %P 2:SCHRITT 293 = A3508 & A4039 + T8 + T9, 3: ST_CON
         IF $OUT[3508] AND $OUT[4039] OR $TIMER_FLAG[8] OR $TIMER_FLAG[9] THEN
            PREV_STEP[9] = APP_INT_STEP[9]
            APP_INT_STEP[9] = 293
         ENDIF
      ;ENDFOLD
   ;ENDFOLD
   ;FOLD SCHRITT 293 -- st. RZ2 Setzhub 2 # Acknowledge -- ;%{P}%MKUKATPVW,%CSTEP,%VST_NR,%P 1:SCHRITT, 2:293, 3: st. RZ2 Setzhub 2 # Acknowledge
      ;FOLD ;%{H}
         Case 293
      ;ENDFOLD
      ;FOLD -- RSK Fehlerausgabe Kraftaufbau -- ;%{SE}%MKUKATPVW %CVW_COM %VCOMMENT %P 2:-- RSK Fehlerausgabe Kraftaufbau --, 3: VW_COMMENT
      ;ENDFOLD
      ;FOLD F325 = !A3508 & T9 ;%{SE}%MKUKATPVW %CVW_SPS %VBOASG %P 2:F325 = !A3508 & T9, 3: BOASG
         $FLAG[325] = NOT $OUT[3508] AND $TIMER_FLAG[9]
      ;ENDFOLD
      ;FOLD F329 = T9 ;%{SE}%MKUKATPVW %CVW_SPS %VBOASG %P 2:F329 = T9, 3: BOASG
         $FLAG[329] = $TIMER_FLAG[9]
      ;ENDFOLD
      ;FOLD -- ServoGun SZ1 oeffnen -- ;%{SE}%MKUKATPVW %CVW_COM %VCOMMENT %P 2:-- ServoGun SZ1 oeffnen --, 3: VW_COMMENT
      ;ENDFOLD
      ;FOLD -- RSK Fehlerausgabe Messen -- ;%{SE}%MKUKATPVW %CVW_COM %VCOMMENT %P 2:-- RSK Fehlerausgabe Messen --, 3: VW_COMMENT
      ;ENDFOLD
      ;FOLD A3510 = AUS ;%{SE}%MKUKATPVW %CVW_SPS %VBOASG %P 2:A3510 = AUS, 3: BOASG
         $OUT[3510] = FALSE
      ;ENDFOLD
      ;FOLD A3514 = AUS ;%{SE}%MKUKATPVW %CVW_SPS %VBOASG %P 2:A3514 = AUS, 3: BOASG
         $OUT[3514] = FALSE
      ;ENDFOLD
      ;FOLD A3512 = EIN ;%{SE}%MKUKATPVW %CVW_SPS %VBOASG %P 2:A3512 = EIN, 3: BOASG
         $OUT[3512] = TRUE
      ;ENDFOLD
      ;FOLD -- Druckvorgabe SK1/ServoGun -- ;%{SE}%MKUKATPVW %CVW_COM %VCOMMENT %P 2:-- Druckvorgabe SK1/ServoGun --, 3: VW_COMMENT
      ;ENDFOLD
      ;FOLD bin4 ( F138 ) = 41 ;%{SE}%MKUKATPVW %CVW_SPS %VARIASG %P 2:bin4 ( F138 ) = 41, 3: ARIASG
         VW(#BINOUT,$FLAG[138],4,41)
      ;ENDFOLD
      ;FOLD bin4 ( F139 ) = 51 ;%{SE}%MKUKATPVW %CVW_SPS %VARIASG %P 2:bin4 ( F139 ) = 51, 3: ARIASG
         VW(#BINOUT,$FLAG[139],4,51)
      ;ENDFOLD
      ;FOLD bin31 ( F138 ) = 41 ;%{SE}%MKUKATPVW %CVW_SPS %VARIASG %P 2:bin31 ( F138 ) = 41, 3: ARIASG
         VW(#BINOUT,$FLAG[138],31,41)
      ;ENDFOLD
      ;FOLD bin31 ( F139 ) = 51 ;%{SE}%MKUKATPVW %CVW_SPS %VARIASG %P 2:bin31 ( F139 ) = 51, 3: ARIASG
         VW(#BINOUT,$FLAG[139],31,51)
      ;ENDFOLD
      ;FOLD -- Wartezeit Programmwechsel SK -- ;%{SE}%MKUKATPVW %CVW_COM %VCOMMENT %P 2:-- Wartezeit Programmwechsel SK --, 3: VW_COMMENT
      ;ENDFOLD
      ;FOLD T8 ( !F334 ) = -2[1/10Sek] ;%{SE}%MKUKATPVW %CVW_SPS %VTASG %P 2:T8 ( !F334 ) = -2[1/10Sek], 3: TASG
         VW(#SET_TIME,NOT $FLAG[334],8,0,-2)
      ;ENDFOLD
      ;FOLD -- Hilfsflag SK Programmwechsel -- ;%{SE}%MKUKATPVW %CVW_COM %VCOMMENT %P 2:-- Hilfsflag SK Programmwechsel --, 3: VW_COMMENT
      ;ENDFOLD
      ;FOLD F334 = EIN ;%{SE}%MKUKATPVW %CVW_SPS %VBOASG %P 2:F334 = EIN, 3: BOASG
         $FLAG[334] = TRUE
      ;ENDFOLD
      ;FOLD SCHRITT 294 = T8 & A4039 & !A3507 ;%{SE}%MKUKATPVW %CVW_SPS %VST_CON %P 2:SCHRITT 294 = T8 & A4039 & !A3507, 3: ST_CON
         IF $TIMER_FLAG[8] AND $OUT[4039] AND NOT $OUT[3507] THEN
            PREV_STEP[9] = APP_INT_STEP[9]
            APP_INT_STEP[9] = 294
         ENDIF
      ;ENDFOLD
   ;ENDFOLD
   ;FOLD SCHRITT 294 -- st. RZ2 Setzhub 2 -- ;%{P}%MKUKATPVW,%CSTEP,%VST_NR,%P 1:SCHRITT, 2:294, 3: st. RZ2 Setzhub 2
      ;FOLD ;%{H}
         Case 294
      ;ENDFOLD
      ;FOLD -- Hilfsflag SK Programmwechsel -- ;%{SE}%MKUKATPVW %CVW_COM %VCOMMENT %P 2:-- Hilfsflag SK Programmwechsel --, 3: VW_COMMENT
      ;ENDFOLD
      ;FOLD F334 = AUS ;%{SE}%MKUKATPVW %CVW_SPS %VBOASG %P 2:F334 = AUS, 3: BOASG
         $FLAG[334] = FALSE
      ;ENDFOLD
      ;FOLD A3512 = AUS ;%{SE}%MKUKATPVW %CVW_SPS %VBOASG %P 2:A3512 = AUS, 3: BOASG
         $OUT[3512] = FALSE
      ;ENDFOLD
      ;FOLD SCHRITT 229 = A4039  & A3506 & A3505 & !A3507 ;%{SE}%MKUKATPVW %CVW_SPS %VST_CON %P 2:SCHRITT 229 = A4039  & A3506 & A3505 & !A3507, 3: ST_CON
         IF $OUT[4039] AND $OUT[3506] AND $OUT[3505] AND NOT $OUT[3507] THEN
            PREV_STEP[9] = APP_INT_STEP[9]
            APP_INT_STEP[9] = 229
         ENDIF
      ;ENDFOLD
   ;ENDFOLD
   ;FOLD SCHRITT 303 -- st. RZ3 # Start-- ;%{P}%MKUKATPVW,%CSTEP,%VST_NR,%P 1:SCHRITT, 2:303, 3: st. RZ3 # Start
      ;FOLD ;%{H}
         Case 303
      ;ENDFOLD
      ;FOLD -- RSK gestartet -- ;%{SE}%MKUKATPVW %CVW_COM %VCOMMENT %P 2:-- RSK gestartet --, 3: VW_COMMENT
      ;ENDFOLD
      ;FOLD F196 = AUS ;%{SE}%MKUKATPVW %CVW_SPS %VBOASG %P 2:F196 = AUS, 3: BOASG
         $FLAG[196] = FALSE
      ;ENDFOLD
      ;FOLD F322 = AUS ;%{SE}%MKUKATPVW %CVW_SPS %VBOASG %P 2:F322 = AUS, 3: BOASG
         $FLAG[322] = FALSE
      ;ENDFOLD
      ;FOLD F323 = AUS ;%{SE}%MKUKATPVW %CVW_SPS %VBOASG %P 2:F323 = AUS, 3: BOASG
         $FLAG[323] = FALSE
      ;ENDFOLD
      ;FOLD F324 = AUS ;%{SE}%MKUKATPVW %CVW_SPS %VBOASG %P 2:F324 = AUS, 3: BOASG
         $FLAG[324] = FALSE
      ;ENDFOLD
      ;FOLD F325 = AUS ;%{SE}%MKUKATPVW %CVW_SPS %VBOASG %P 2:F325 = AUS, 3: BOASG
         $FLAG[325] = FALSE
      ;ENDFOLD
      ;FOLD F326 = AUS ;%{SE}%MKUKATPVW %CVW_SPS %VBOASG %P 2:F326 = AUS, 3: BOASG
         $FLAG[326] = FALSE
      ;ENDFOLD
      ;FOLD F327 = AUS ;%{SE}%MKUKATPVW %CVW_SPS %VBOASG %P 2:F327 = AUS, 3: BOASG
         $FLAG[327] = FALSE
      ;ENDFOLD
      ;FOLD F329 = AUS ;%{SE}%MKUKATPVW %CVW_SPS %VBOASG %P 2:F329 = AUS, 3: BOASG
         $FLAG[329] = FALSE
      ;ENDFOLD
      ;FOLD -- ServoGun SZ1 Zaehler -- ;%{SE}%MKUKATPVW %CVW_COM %VCOMMENT %P 2:-- ServoGun SZ1 Zaehler --, 3: VW_COMMENT
      ;ENDFOLD
      ;FOLD F186 = AUS ;%{SE}%MKUKATPVW %CVW_SPS %VBOASG %P 2:F186 = AUS, 3: BOASG
         $FLAG[186] = FALSE
      ;ENDFOLD
      ;FOLD F187 = AUS ;%{SE}%MKUKATPVW %CVW_SPS %VBOASG %P 2:F187 = AUS, 3: BOASG
         $FLAG[187] = FALSE
      ;ENDFOLD
      ;FOLD F188 = AUS ;%{SE}%MKUKATPVW %CVW_SPS %VBOASG %P 2:F188 = AUS, 3: BOASG
         $FLAG[188] = FALSE
      ;ENDFOLD
      ;FOLD F189 = AUS ;%{SE}%MKUKATPVW %CVW_SPS %VBOASG %P 2:F189 = AUS, 3: BOASG
         $FLAG[189] = FALSE
      ;ENDFOLD
      ;FOLD F190 = AUS ;%{SE}%MKUKATPVW %CVW_SPS %VBOASG %P 2:F190 = AUS, 3: BOASG
         $FLAG[190] = FALSE
      ;ENDFOLD
      ;FOLD F191 = AUS ;%{SE}%MKUKATPVW %CVW_SPS %VBOASG %P 2:F191 = AUS, 3: BOASG
         $FLAG[191] = FALSE
      ;ENDFOLD
      ;FOLD -- Hilfsflags Funktionstest KF Motor -- ;%{SE}%MKUKATPVW %CVW_COM %VCOMMENT %P 2:-- Hilfsflags Funktionstest KF Motor --, 3: VW_COMMENT
      ;ENDFOLD
      ;FOLD F312 = AUS ;%{SE}%MKUKATPVW %CVW_SPS %VBOASG %P 2:F312 = AUS, 3: BOASG
         $FLAG[312] = FALSE
      ;ENDFOLD
      ;FOLD F313 = AUS ;%{SE}%MKUKATPVW %CVW_SPS %VBOASG %P 2:F313 = AUS, 3: BOASG
         $FLAG[313] = FALSE
      ;ENDFOLD
      ;FOLD -- Hilfsflags ServoGun Start -- ;%{SE}%MKUKATPVW %CVW_COM %VCOMMENT %P 2:-- Hilfsflags ServoGun Start --, 3: VW_COMMENT
      ;ENDFOLD
      ;FOLD F276 = EIN ;%{SE}%MKUKATPVW %CVW_SPS %VBOASG %P 2:F276 = EIN, 3: BOASG
         $FLAG[276] = TRUE
      ;ENDFOLD
      ;FOLD A3935 = AUS ;%{SE}%MKUKATPVW %CVW_SPS %VBOASG %P 2:A3935 = AUS, 3: BOASG
         $OUT[3935] = FALSE
      ;ENDFOLD
      ;FOLD A3936 = AUS ;%{SE}%MKUKATPVW %CVW_SPS %VBOASG %P 2:A3936 = AUS, 3: BOASG
         $OUT[3936] = FALSE
      ;ENDFOLD
      ;FOLD A3510 = EIN ;%{SE}%MKUKATPVW %CVW_SPS %VBOASG %P 2:A3510 = EIN, 3: BOASG
         $OUT[3510] = TRUE
      ;ENDFOLD
      ;FOLD A3511 = AUS ;%{SE}%MKUKATPVW %CVW_SPS %VBOASG %P 2:A3511 = AUS, 3: BOASG
         $OUT[3511] = FALSE
      ;ENDFOLD
      ;FOLD A3514 = AUS ;%{SE}%MKUKATPVW %CVW_SPS %VBOASG %P 2:A3514 = AUS, 3: BOASG
         $OUT[3514] = FALSE
      ;ENDFOLD
      ;FOLD A3513 = AUS ;%{SE}%MKUKATPVW %CVW_SPS %VBOASG %P 2:A3513 = AUS, 3: BOASG
         $OUT[3513] = FALSE
      ;ENDFOLD
      ;FOLD A3512 = AUS ;%{SE}%MKUKATPVW %CVW_SPS %VBOASG %P 2:A3512 = AUS, 3: BOASG
         $OUT[3512] = FALSE
      ;ENDFOLD
      ;FOLD -- Hilfsflags ServoGun Ende -- ;%{SE}%MKUKATPVW %CVW_COM %VCOMMENT %P 2:-- Hilfsflags ServoGun Ende --, 3: VW_COMMENT
      ;ENDFOLD
      ;FOLD -- Ausblasen zuruecksetzen -- ;%{SE}%MKUKATPVW %CVW_COM %VCOMMENT %P 2:-- Ausblasen zuruecksetzen --, 3: VW_COMMENT
      ;ENDFOLD
      ;FOLD A836 = AUS ;%{SE}%MKUKATPVW %CVW_SPS %VBOASG %P 2:A836 = AUS, 3: BOASG
         $OUT[836] = FALSE
      ;ENDFOLD
      ;FOLD A996 = AUS ;%{SE}%MKUKATPVW %CVW_SPS %VBOASG %P 2:A996 = AUS, 3: BOASG
         $OUT[996] = FALSE
      ;ENDFOLD
      ;FOLD A1156 = AUS ;%{SE}%MKUKATPVW %CVW_SPS %VBOASG %P 2:A1156 = AUS, 3: BOASG
         $OUT[1156] = FALSE
      ;ENDFOLD
      ;FOLD -- Prognummer setzen -- ;%{SE}%MKUKATPVW %CVW_COM %VCOMMENT %P 2:-- Prognummer setzen --, 3: VW_COMMENT
      ;ENDFOLD
      ;FOLD bin28 ( EIN ) = 0 ;%{SE}%MKUKATPVW %CVW_SPS %VARIASG %P 2:bin28 ( EIN ) = 0, 3: ARIASG
         VW(#BINOUT,TRUE,28,0)
      ;ENDFOLD
      ;FOLD bin9 ( EIN ) = 31 ;%{SE}%MKUKATPVW %CVW_SPS %VARIASG %P 2:bin9 ( EIN ) = 31, 3: ARIASG
         VW(#BINOUT,TRUE,9,31)
      ;ENDFOLD
      ;FOLD bin30 ( EIN ) = p113 ;%{SE}%MKUKATPVW %CVW_SPS %VARIASG %P 2:bin30 ( EIN ) = p113, 3: ARIASG
         VW(#BINOUT,TRUE,30,PROCPAR[113])
      ;ENDFOLD
      ;FOLD bin31 ( EIN ) = 31 ;%{SE}%MKUKATPVW %CVW_SPS %VARIASG %P 2:bin31 ( EIN ) = 31, 3: ARIASG
         VW(#BINOUT,TRUE,31,31)
      ;ENDFOLD
      ;FOLD -- Wartezeit Programmwechsel SK -- ;%{SE}%MKUKATPVW %CVW_COM %VCOMMENT %P 2:-- Wartezeit Programmwechsel SK --, 3: VW_COMMENT
      ;ENDFOLD
      ;FOLD T8 ( !F334 ) = -2[1/10Sek] ;%{SE}%MKUKATPVW %CVW_SPS %VTASG %P 2:T8 ( !F334 ) = -2[1/10Sek], 3: TASG
         VW(#SET_TIME,NOT $FLAG[334],8,0,-2)
      ;ENDFOLD
      ;FOLD -- Hilfsflag SK Programmwechsel -- ;%{SE}%MKUKATPVW %CVW_COM %VCOMMENT %P 2:-- Hilfsflag SK Programmwechsel --, 3: VW_COMMENT
      ;ENDFOLD
      ;FOLD F334 = EIN ;%{SE}%MKUKATPVW %CVW_SPS %VBOASG %P 2:F334 = EIN, 3: BOASG
         $FLAG[334] = TRUE
      ;ENDFOLD
      ;FOLD -- Stat. ServoGun SZ1 beim Fraesen -- ;%{SE}%MKUKATPVW %CVW_COM %VCOMMENT %P 2:-- Stat. ServoGun SZ1 beim Fraesen --, 3: VW_COMMENT
      ;ENDFOLD
      ;FOLD A116 = EIN ;%{SE}%MKUKATPVW %CVW_SPS %VBOASG %P 2:A116 = EIN, 3: BOASG
         $OUT[116] = TRUE
      ;ENDFOLD
      ;FOLD A192 = EIN ;%{SE}%MKUKATPVW %CVW_SPS %VBOASG %P 2:A192 = EIN, 3: BOASG
         $OUT[192] = TRUE
      ;ENDFOLD
      ;FOLD -- Quitt. Fraesen SK1 AUS -- ;%{SE}%MKUKATPVW %CVW_COM %VCOMMENT %P 2:-- Quitt. Fraesen SK1 AUS --, 3: VW_COMMENT
      ;ENDFOLD
      ;FOLD A1106 = F830 ;%{SE}%MKUKATPVW %CVW_SPS %VBOASG %P 2:A1106 = F830, 3: BOASG
         $OUT[1106] = $FLAG[830]
      ;ENDFOLD
      ;FOLD A1042 = !F830 ;%{SE}%MKUKATPVW %CVW_SPS %VBOASG %P 2:A1042 = !F830, 3: BOASG
         $OUT[1042] = NOT $FLAG[830]
      ;ENDFOLD
      ;FOLD SCHRITT 304 = T8 & A4039 ;%{SE}%MKUKATPVW %CVW_SPS %VST_CON %P 2:SCHRITT 304 = T8 & A4039, 3: ST_CON
         IF $TIMER_FLAG[8] AND $OUT[4039] THEN
            PREV_STEP[9] = APP_INT_STEP[9]
            APP_INT_STEP[9] = 304
         ENDIF
      ;ENDFOLD
   ;ENDFOLD
   ;FOLD SCHRITT 304 -- st. RZ3 -- ;%{P}%MKUKATPVW,%CSTEP,%VST_NR,%P 1:SCHRITT, 2:304, 3: st. RZ3
      ;FOLD ;%{H}
         Case 304
      ;ENDFOLD
      ;FOLD -- Hilfsflag SK Programmwechsel -- ;%{SE}%MKUKATPVW %CVW_COM %VCOMMENT %P 2:-- Hilfsflag SK Programmwechsel --, 3: VW_COMMENT
      ;ENDFOLD
      ;FOLD F334 = AUS ;%{SE}%MKUKATPVW %CVW_SPS %VBOASG %P 2:F334 = AUS, 3: BOASG
         $FLAG[334] = FALSE
      ;ENDFOLD
      ;FOLD -- Ueberwachungszeit KF1 EIN -- ;%{SE}%MKUKATPVW %CVW_COM %VCOMMENT %P 2:-- Ueberwachungszeit KF1 EIN --, 3: VW_COMMENT
      ;ENDFOLD
      ;FOLD T7 ( EIN ) = -50[1/10Sek] ;%{SE}%MKUKATPVW %CVW_SPS %VTASG %P 2:T7 ( EIN ) = -50[1/10Sek], 3: TASG
         VW(#SET_TIME,TRUE,7,0,-50)
      ;ENDFOLD
      ;FOLD -- KF1 einschalten -- ;%{SE}%MKUKATPVW %CVW_COM %VCOMMENT %P 2:-- KF1 einschalten --, 3: VW_COMMENT
      ;ENDFOLD
      ;FOLD i1 (EIN) = 0 ;%{SE}%MKUKATPVW %CVW_SPS %VARIASG %P 2:i1 (EIN) = 0, 3: ARIASG
         VW(#COUNTER,TRUE,1,0)
      ;ENDFOLD
      ;FOLD A1154 = EIN ;%{SE}%MKUKATPVW %CVW_SPS %VBOASG %P 2:A1154 = EIN, 3: BOASG
         $OUT[1154] = TRUE
      ;ENDFOLD
      ;FOLD SCHRITT 305 = A4039 ;%{SE}%MKUKATPVW %CVW_SPS %VST_CON %P 2:SCHRITT 305 = A4039, 3: ST_CON
         IF $OUT[4039] THEN
            PREV_STEP[9] = APP_INT_STEP[9]
            APP_INT_STEP[9] = 305
         ENDIF
      ;ENDFOLD
   ;ENDFOLD
   ;FOLD SCHRITT 305 -- st. RZ3 # Funktionstest KF -- ;%{P}%MKUKATPVW,%CSTEP,%VST_NR,%P 1:SCHRITT, 2:305, 3: st. RZ3 # Funktionstest KF
      ;FOLD ;%{H}
         Case 305
      ;ENDFOLD
      ;FOLD -- Funktionstest KF Motor -- ;%{SE}%MKUKATPVW %CVW_COM %VCOMMENT %P 2:-- Funktionstest KF Motor --, 3: VW_COMMENT
      ;ENDFOLD
      ;FOLD F312 = EIN ;%{SE}%MKUKATPVW %CVW_SPS %VBOASG %P 2:F312 = EIN, 3: BOASG
         $FLAG[312] = TRUE
      ;ENDFOLD
      ;FOLD F313 = i1 > 2 ;%{SE}%MKUKATPVW %CVW_SPS %VBOCMP %P 2:F313 = i1 > 2, 3: BOCMP
         $FLAG[313] = $COUNT_I[1] > 2
      ;ENDFOLD
      ;FOLD SCHRITT 306 = (F313 + T7) & A4039 ;%{SE}%MKUKATPVW %CVW_SPS %VST_CON %P 2:SCHRITT 306 = (F313 + T7) & A4039, 3: ST_CON
         IF ($FLAG[313] OR $TIMER_FLAG[7]) AND $OUT[4039] THEN
            PREV_STEP[9] = APP_INT_STEP[9]
            APP_INT_STEP[9] = 306
         ENDIF
      ;ENDFOLD
   ;ENDFOLD
   ;FOLD SCHRITT 306 -- st. RZ3 -- ;%{P}%MKUKATPVW,%CSTEP,%VST_NR,%P 1:SCHRITT, 2:306, 3: st. RZ3
      ;FOLD ;%{H}
         Case 306
      ;ENDFOLD
      ;FOLD F312 = AUS ;%{SE}%MKUKATPVW %CVW_SPS %VBOASG %P 2:F312 = AUS, 3: BOASG
         $FLAG[312] = FALSE
      ;ENDFOLD
      ;FOLD -- Ueberwachungszeit KS1 schwenken -- ;%{SE}%MKUKATPVW %CVW_COM %VCOMMENT %P 2:-- Ueberwachungszeit KS1 schwenken --, 3: VW_COMMENT
      ;ENDFOLD
      ;FOLD t8 ( EIN ) = -100[1/10Sek] ;%{SE}%MKUKATPVW %CVW_SPS %VTASG %P 2:t8 ( EIN ) = -100[1/10Sek], 3: TASG
         VW(#SET_TIME,TRUE,8,0,-100)
      ;ENDFOLD
      ;FOLD SCHRITT 307 = A4039 ;%{SE}%MKUKATPVW %CVW_SPS %VST_CON %P 2:SCHRITT 307 = A4039, 3: ST_CON
         IF $OUT[4039] THEN
            PREV_STEP[9] = APP_INT_STEP[9]
            APP_INT_STEP[9] = 307
         ENDIF
      ;ENDFOLD
   ;ENDFOLD
   ;FOLD SCHRITT 307 -- st. RZ3 # Fehler KF -- ;%{P}%MKUKATPVW,%CSTEP,%VST_NR,%P 1:SCHRITT, 2:307, 3: st. RZ3 # Fehler KF
      ;FOLD ;%{H}
         Case 307
      ;ENDFOLD
      ;FOLD -- RSK Fehlerausgabe KF1 Initiator/Motor -- ;%{SE}%MKUKATPVW %CVW_COM %VCOMMENT %P 2:-- RSK Fehlerausgabe KF1 Initiator/Motor --, 3: VW_COMMENT
      ;ENDFOLD
      ;FOLD F322 = !F313 ;%{SE}%MKUKATPVW %CVW_SPS %VBOASG %P 2:F322 = !F313, 3: BOASG
         $FLAG[322] = NOT $FLAG[313]
      ;ENDFOLD
      ;FOLD -- RSK Fehlerausgabe KS1 Ruhest. -- ;%{SE}%MKUKATPVW %CVW_COM %VCOMMENT %P 2:-- RSK Fehlerausgabe KS1 Ruhest. --, 3: VW_COMMENT
      ;ENDFOLD
      ;FOLD F323 = (!E1156 + E1157 + E1158 + !E1159) & !F324 & !F328 ;%{SE}%MKUKATPVW %CVW_SPS %VBOASG %P 2:F323 = (!E1156 + E1157 + E1158 + !E1159) & !F324 & !F328, 3: BOASG
         $FLAG[323] = (NOT $IN[1156] OR $IN[1157] OR $IN[1158] OR NOT $IN[1159]) AND NOT $FLAG[324] AND NOT $FLAG[328]
      ;ENDFOLD
      ;FOLD -- RSK Sammelstoerung -- ;%{SE}%MKUKATPVW %CVW_COM %VCOMMENT %P 2:-- RSK Sammelstoerung --, 3: VW_COMMENT
      ;ENDFOLD
      ;FOLD F329 = F322 + F323 + T8 ;%{SE}%MKUKATPVW %CVW_SPS %VBOASG %P 2:F329 = F322 + F323 + T8, 3: BOASG
         $FLAG[329] = $FLAG[322] OR $FLAG[323] OR $TIMER_FLAG[8]
      ;ENDFOLD
      ;FOLD T7 ( EIN ) = STOP ;%{SE}%MKUKATPVW %CVW_SPS %VTSTOP %P 2:T7 ( EIN ) = STOP, 3: TSTOP
         VW(#SET_TIME,TRUE,7,1,0)
      ;ENDFOLD
      ;FOLD -- KF Motor Ein -- ;%{SE}%MKUKATPVW %CVW_COM %VCOMMENT %P 2:-- KF Motor Ein --, 3: VW_COMMENT
      ;ENDFOLD
      ;FOLD A1154 = !F322 & !F323 ;%{SE}%MKUKATPVW %CVW_SPS %VBOASG %P 2:A1154 = !F322 & !F323, 3: BOASG
         $OUT[1154] = NOT $FLAG[322] AND NOT $FLAG[323]
      ;ENDFOLD
      ;FOLD -- KF1 Versetzeinheit vor -- ;%{SE}%MKUKATPVW %CVW_COM %VCOMMENT %P 2:-- KF1 Versetzeinheit vor --, 3: VW_COMMENT
      ;ENDFOLD
      ;FOLD A1155 = !F322 & !F323 & F564 ;%{SE}%MKUKATPVW %CVW_SPS %VBOASG %P 2:A1155 = !F322 & !F323 & F564, 3: BOASG
         $OUT[1155] = NOT $FLAG[322] AND NOT $FLAG[323] AND $FLAG[564]
      ;ENDFOLD
      ;FOLD SCHRITT 308 = (!F322 & !F323) & (E1155 & F564 + !E1155 & !F564) & A4039 ;%{SE}%MKUKATPVW %CVW_SPS %VST_CON %P 2:SCHRITT 308 = (!F322 & !F323) & (E1155 & F564 + !E1155 & !F564) & A4039, 3: ST_CON
         IF (NOT $FLAG[322] AND NOT $FLAG[323]) AND ($IN[1155] AND $FLAG[564] OR NOT $IN[1155] AND NOT $FLAG[564]) AND $OUT[4039] THEN
            PREV_STEP[9] = APP_INT_STEP[9]
            APP_INT_STEP[9] = 308
         ENDIF
      ;ENDFOLD
      ;FOLD SCHRITT 334 = (F322 + F323) & !F324 & !F328 & A4039 & (E26 + E27) ;%{SE}%MKUKATPVW %CVW_SPS %VST_CON %P 2:SCHRITT 334 = (F322 + F323) & !F324 & !F328 & A4039 & (E26 + E27), 3: ST_CON
         IF ($FLAG[322] OR $FLAG[323]) AND NOT $FLAG[324] AND NOT $FLAG[328] AND $OUT[4039] AND ($IN[26] OR $IN[27]) THEN
            PREV_STEP[9] = APP_INT_STEP[9]
            APP_INT_STEP[9] = 334
         ENDIF
      ;ENDFOLD
   ;ENDFOLD
   ;FOLD SCHRITT 308 -- st. RZ3 # Sicherheit KF -- ;%{P}%MKUKATPVW,%CSTEP,%VST_NR,%P 1:SCHRITT, 2:308, 3: st. RZ3 # Sicherheit KF
      ;FOLD ;%{H}
         Case 308
      ;ENDFOLD
      ;FOLD -- RSK Sammelstoerung -- ;%{SE}%MKUKATPVW %CVW_COM %VCOMMENT %P 2:-- RSK Sammelstoerung --, 3: VW_COMMENT
      ;ENDFOLD
      ;FOLD F329 = AUS ;%{SE}%MKUKATPVW %CVW_SPS %VBOASG %P 2:F329 = AUS, 3: BOASG
         $FLAG[329] = FALSE
      ;ENDFOLD
      ;FOLD F324 = AUS ;%{SE}%MKUKATPVW %CVW_SPS %VBOASG %P 2:F324 = AUS, 3: BOASG
         $FLAG[324] = FALSE
      ;ENDFOLD
      ;FOLD F328 = AUS ;%{SE}%MKUKATPVW %CVW_SPS %VBOASG %P 2:F328 = AUS, 3: BOASG
         $FLAG[328] = FALSE
      ;ENDFOLD
      ;FOLD -- Wartebedingung schwenken -- ;%{SE}%MKUKATPVW %CVW_COM %VCOMMENT %P 2:-- Wartebedingung schwenken --, 3: VW_COMMENT
      ;ENDFOLD
      ;FOLD SCHRITT 309 = A3926 & A4039 ;%{SE}%MKUKATPVW %CVW_SPS %VST_CON %P 2:SCHRITT 309 = A3926 & A4039, 3: ST_CON
         IF $OUT[3926] AND $OUT[4039] THEN
            PREV_STEP[9] = APP_INT_STEP[9]
            APP_INT_STEP[9] = 309
         ENDIF
      ;ENDFOLD
   ;ENDFOLD
   ;FOLD SCHRITT 309 -- st. RZ3 # KS in AS schwenken -- ;%{P}%MKUKATPVW,%CSTEP,%VST_NR,%P 1:SCHRITT, 2:309, 3: st. RZ3 # KS in AS schwenken
      ;FOLD ;%{H}
         Case 309
      ;ENDFOLD
      ;FOLD -- KS1 in Arbeitsstellung schwenken -- ;%{SE}%MKUKATPVW %CVW_COM %VCOMMENT %P 2:-- KS1 in Arbeitsstellung schwenken --, 3: VW_COMMENT
      ;ENDFOLD
      ;FOLD A1160 = A3926 & !E1157 & (E1155 & F564 + !E1155 & !F564) ;%{SE}%MKUKATPVW %CVW_SPS %VBOASG %P 2:A1160 = A3926 & !E1157 & (E1155 & F564 + !E1155 & !F564), 3: BOASG
         $OUT[1160] = $OUT[3926] AND NOT $IN[1157] AND ($IN[1155] AND $FLAG[564] OR NOT $IN[1155] AND NOT $FLAG[564])
      ;ENDFOLD
      ;FOLD -- KF1 Ausblasen -- ;%{SE}%MKUKATPVW %CVW_COM %VCOMMENT %P 2:-- KF1 Ausblasen --, 3: VW_COMMENT
      ;ENDFOLD
      ;FOLD A1156 = F330 + !F330 & !F331 & !F332 ;%{SE}%MKUKATPVW %CVW_SPS %VBOASG %P 2:A1156 = F330 + !F330 & !F331 & !F332, 3: BOASG
         $OUT[1156] = $FLAG[330] OR NOT $FLAG[330] AND NOT $FLAG[331] AND NOT $FLAG[332]
      ;ENDFOLD
      ;FOLD SCHRITT 310 =  A3926 & (A1160 + E1157 + T8) & A4039 ;%{SE}%MKUKATPVW %CVW_SPS %VST_CON %P 2:SCHRITT 310 =  A3926 & (A1160 + E1157 + T8) & A4039, 3: ST_CON
         IF $OUT[3926] AND ($OUT[1160] OR $IN[1157] OR $TIMER_FLAG[8]) AND $OUT[4039] THEN
            PREV_STEP[9] = APP_INT_STEP[9]
            APP_INT_STEP[9] = 310
         ENDIF
      ;ENDFOLD
   ;ENDFOLD
   ;FOLD SCHRITT 310 -- st. RZ3 -- ;%{P}%MKUKATPVW,%CSTEP,%VST_NR,%P 1:SCHRITT, 2:310, 3: st. RZ3
      ;FOLD ;%{H}
         Case 310
      ;ENDFOLD
      ;FOLD -- RSK Fehlerausgabe KF Versetzeinheit -- ;%{SE}%MKUKATPVW %CVW_COM %VCOMMENT %P 2:-- RSK Fehlerausgabe KF Versetzeinheit --, 3: VW_COMMENT
      ;ENDFOLD
      ;FOLD F328 = !E1155 & F564 & !F324 ;%{SE}%MKUKATPVW %CVW_SPS %VBOASG %P 2:F328 = !E1155 & F564 & !F324, 3: BOASG
         $FLAG[328] = NOT $IN[1155] AND $FLAG[564] AND NOT $FLAG[324]
      ;ENDFOLD
      ;FOLD -- RSK Fehlerausgabe KS1 Arbeitsstellung -- ;%{SE}%MKUKATPVW %CVW_COM %VCOMMENT %P 2:-- RSK Fehlerausgabe KS1 Arbeitsstellung --, 3: VW_COMMENT
      ;ENDFOLD
      ;FOLD F324 = (E1156 + !E1157 + !E1158 + E1159) & T8 & (E1155 + !F564) + F324 ;%{SE}%MKUKATPVW %CVW_SPS %VBOASG %P 2:F324 = (E1156 + !E1157 + !E1158 + E1159) & T8 & (E1155 + !F564) + F324, 3: BOASG
         $FLAG[324] = ($IN[1156] OR NOT $IN[1157] OR NOT $IN[1158] OR $IN[1159]) AND $TIMER_FLAG[8] AND ($IN[1155] OR NOT $FLAG[564]) OR $FLAG[324]
      ;ENDFOLD
      ;FOLD -- RSK Fehlerausgabe EZ/SP min. Oeffnung -- ;%{SE}%MKUKATPVW %CVW_COM %VCOMMENT %P 2:-- RSK Fehlerausgabe EZ/SP min. Oeffnung --, 3: VW_COMMENT
      ;ENDFOLD
      ;FOLD F333 = !A3926 ;%{SE}%MKUKATPVW %CVW_SPS %VBOASG %P 2:F333 = !A3926, 3: BOASG
         $FLAG[333] = NOT $OUT[3926]
      ;ENDFOLD
      ;FOLD -- RSK Sammelstoerung -- ;%{SE}%MKUKATPVW %CVW_COM %VCOMMENT %P 2:-- RSK Sammelstoerung --, 3: VW_COMMENT
      ;ENDFOLD
      ;FOLD F329 = F324 + F328 + F333 ;%{SE}%MKUKATPVW %CVW_SPS %VBOASG %P 2:F329 = F324 + F328 + F333, 3: BOASG
         $FLAG[329] = $FLAG[324] OR $FLAG[328] OR $FLAG[333]
      ;ENDFOLD
      ;FOLD A1154 = !F324 & !F328 ;%{SE}%MKUKATPVW %CVW_SPS %VBOASG %P 2:A1154 = !F324 & !F328, 3: BOASG
         $OUT[1154] = NOT $FLAG[324] AND NOT $FLAG[328]
      ;ENDFOLD
      ;FOLD -- KF1 Ausblasen -- ;%{SE}%MKUKATPVW %CVW_COM %VCOMMENT %P 2:-- KF1 Ausblasen --, 3: VW_COMMENT
      ;ENDFOLD
      ;FOLD A1156 = (F330 + !F330 & !F331 & !F332) & !F324 & !F328 ;%{SE}%MKUKATPVW %CVW_SPS %VBOASG %P 2:A1156 = (F330 + !F330 & !F331 & !F332) & !F324 & !F328, 3: BOASG
         $OUT[1156] = ($FLAG[330] OR NOT $FLAG[330] AND NOT $FLAG[331] AND NOT $FLAG[332]) AND NOT $FLAG[324] AND NOT $FLAG[328]
      ;ENDFOLD
      ;FOLD A1155 = F564 ;%{SE}%MKUKATPVW %CVW_SPS %VBOASG %P 2:A1155 = F564, 3: BOASG
         $OUT[1155] = $FLAG[564]
      ;ENDFOLD
      ;FOLD -- Verweilzeit Versetzeinheit Rueck -- ;%{SE}%MKUKATPVW %CVW_COM %VCOMMENT %P 2:-- Verweilzeit Versetzeinheit Rueck --, 3: VW_COMMENT
      ;ENDFOLD
      ;FOLD t11 ( EIN ) = i24[1/10Sek] ;%{SE}%MKUKATPVW %CVW_SPS %VTASG %P 2:t11 ( EIN ) = i24[1/10Sek], 3: TASG
         VW(#SET_TIME,TRUE,11,0,$COUNT_I[24])
      ;ENDFOLD
      ;FOLD SCHRITT 303 = (F324 + F328) & (E26 + E27) & A4039 ;%{SE}%MKUKATPVW %CVW_SPS %VST_CON %P 2:SCHRITT 303 = (F324 + F328) & (E26 + E27) & A4039, 3: ST_CON
         IF ($FLAG[324] OR $FLAG[328]) AND ($IN[26] OR $IN[27]) AND $OUT[4039] THEN
            PREV_STEP[9] = APP_INT_STEP[9]
            APP_INT_STEP[9] = 303
         ENDIF
      ;ENDFOLD
      ;FOLD SCHRITT 311 = !F324 & !F328 & !E1156 & E1157 & E1158 & !E1159 & A4039 ;%{SE}%MKUKATPVW %CVW_SPS %VST_CON %P 2:SCHRITT 311 = !F324 & !F328 & !E1156 & E1157 & E1158 & !E1159 & A4039, 3: ST_CON
         IF NOT $FLAG[324] AND NOT $FLAG[328] AND NOT $IN[1156] AND $IN[1157] AND $IN[1158] AND NOT $IN[1159] AND $OUT[4039] THEN
            PREV_STEP[9] = APP_INT_STEP[9]
            APP_INT_STEP[9] = 311
         ENDIF
      ;ENDFOLD
   ;ENDFOLD
   ;FOLD SCHRITT 311 -- st. RZ3 -- ;%{P}%MKUKATPVW,%CSTEP,%VST_NR,%P 1:SCHRITT, 2:311, 3: st. RZ3
      ;FOLD ;%{H}
         Case 311
      ;ENDFOLD
      ;FOLD -- Umdreh. KF setzen zwischenspeichern -- ;%{SE}%MKUKATPVW %CVW_COM %VCOMMENT %P 2:-- Umdreh. KF setzen zwischenspeichern --, 3: VW_COMMENT
      ;ENDFOLD
      ;FOLD i45 ( EIN ) = i19 ;%{SE}%MKUKATPVW %CVW_SPS %VARIASG %P 2:i45 ( EIN ) = i19, 3: ARIASG
         VW(#COUNTER,TRUE,45,$COUNT_I[19])
      ;ENDFOLD
      ;FOLD i19 ( F191 ) = i44 ;%{SE}%MKUKATPVW %CVW_SPS %VARIASG %P 2:i19 ( F191 ) = i44, 3: ARIASG
         VW(#COUNTER,$FLAG[191],19,$COUNT_I[44])
      ;ENDFOLD
      ;FOLD i1 ( EIN ) = 0 ;%{SE}%MKUKATPVW %CVW_SPS %VARIASG %P 2:i1 ( EIN ) = 0, 3: ARIASG
         VW(#COUNTER,TRUE,1,0)
      ;ENDFOLD
      ;FOLD F190 = AUS ;%{SE}%MKUKATPVW %CVW_SPS %VBOASG %P 2:F190 = AUS, 3: BOASG
         $FLAG[190] = FALSE
      ;ENDFOLD
      ;FOLD F312 = AUS ;%{SE}%MKUKATPVW %CVW_SPS %VBOASG %P 2:F312 = AUS, 3: BOASG
         $FLAG[312] = FALSE
      ;ENDFOLD
      ;FOLD F313 = AUS ;%{SE}%MKUKATPVW %CVW_SPS %VBOASG %P 2:F313 = AUS, 3: BOASG
         $FLAG[313] = FALSE
      ;ENDFOLD
      ;FOLD F324 = AUS ;%{SE}%MKUKATPVW %CVW_SPS %VBOASG %P 2:F324 = AUS, 3: BOASG
         $FLAG[324] = FALSE
      ;ENDFOLD
      ;FOLD F328 = AUS ;%{SE}%MKUKATPVW %CVW_SPS %VBOASG %P 2:F328 = AUS, 3: BOASG
         $FLAG[328] = FALSE
      ;ENDFOLD
      ;FOLD -- ServoGun Dress in Positon AUS -- ;%{SE}%MKUKATPVW %CVW_COM %VCOMMENT %P 2:-- ServoGun Dress in Positon AUS --, 3: VW_COMMENT
      ;ENDFOLD
      ;FOLD A3871 = AUS ;%{SE}%MKUKATPVW %CVW_SPS %VBOASG %P 2:A3871 = AUS, 3: BOASG
         $OUT[3871] = FALSE
      ;ENDFOLD
      ;FOLD -- KF1 einschalten nach Fehler -- ;%{SE}%MKUKATPVW %CVW_COM %VCOMMENT %P 2:-- KF1 einschalten nach Fehler --, 3: VW_COMMENT
      ;ENDFOLD
      ;FOLD A1154 = EIN ;%{SE}%MKUKATPVW %CVW_SPS %VBOASG %P 2:A1154 = EIN, 3: BOASG
         $OUT[1154] = TRUE
      ;ENDFOLD
      ;FOLD -- KF1 Versetzeinheit rueck -- ;%{SE}%MKUKATPVW %CVW_COM %VCOMMENT %P 2:-- KF1 Versetzeinheit rueck --, 3: VW_COMMENT
      ;ENDFOLD
      ;FOLD A1155 = AUS ;%{SE}%MKUKATPVW %CVW_SPS %VBOASG %P 2:A1155 = AUS, 3: BOASG
         $OUT[1155] = FALSE
      ;ENDFOLD
      ;FOLD bin30 ( EIN ) = p113 ;%{SE}%MKUKATPVW %CVW_SPS %VARIASG %P 2:bin30 ( EIN ) = p113, 3: ARIASG
         VW(#BINOUT,TRUE,30,PROCPAR[113])
      ;ENDFOLD
      ;FOLD SCHRITT 312 = T11 & A4039 ;%{SE}%MKUKATPVW %CVW_SPS %VST_CON %P 2:SCHRITT 312 = T11 & A4039, 3: ST_CON
         IF $TIMER_FLAG[11] AND $OUT[4039] THEN
            PREV_STEP[9] = APP_INT_STEP[9]
            APP_INT_STEP[9] = 312
         ENDIF
      ;ENDFOLD
   ;ENDFOLD
   ;FOLD SCHRITT 312 -- st. RZ3 -- ;%{P}%MKUKATPVW,%CSTEP,%VST_NR,%P 1:SCHRITT, 2:312, 3: st. RZ3
      ;FOLD ;%{H}
         Case 312
      ;ENDFOLD
      ;FOLD -- Ueberwachungszeit ServoGun SZ1 schliessen -- ;%{SE}%MKUKATPVW %CVW_COM %VCOMMENT %P 2:-- Ueberwachungszeit ServoGun SZ1 schliessen --, 3: VW_COMMENT
      ;ENDFOLD
      ;FOLD t9 ( EIN ) = -80[1/10Sek] ;%{SE}%MKUKATPVW %CVW_SPS %VTASG %P 2:t9 ( EIN ) = -80[1/10Sek], 3: TASG
         VW(#SET_TIME,TRUE,9,0,-80)
      ;ENDFOLD
      ;FOLD -- Warte bis Fraeser in Position -- ;%{SE}%MKUKATPVW %CVW_COM %VCOMMENT %P 2:-- Warte bis Fraeser in Position --, 3: VW_COMMENT
      ;ENDFOLD
      ;FOLD SCHRITT 313 = !E1156 & E1157 & E1158 & !E1159 & A4039 ;%{SE}%MKUKATPVW %CVW_SPS %VST_CON %P 2:SCHRITT 313 = !E1156 & E1157 & E1158 & !E1159 & A4039, 3: ST_CON
         IF NOT $IN[1156] AND $IN[1157] AND $IN[1158] AND NOT $IN[1159] AND $OUT[4039] THEN
            PREV_STEP[9] = APP_INT_STEP[9]
            APP_INT_STEP[9] = 313
         ENDIF
      ;ENDFOLD
   ;ENDFOLD
   ;FOLD SCHRITT 313 -- st. RZ3 # DressInPos -- ;%{P}%MKUKATPVW,%CSTEP,%VST_NR,%P 1:SCHRITT, 2:313, 3: st. RZ3 # DressInPos
      ;FOLD ;%{H}
         Case 313
      ;ENDFOLD
      ;FOLD t11 ( EIN ) = STOP ;%{SE}%MKUKATPVW %CVW_SPS %VTSTOP %P 2:t11 ( EIN ) = STOP, 3: TSTOP
         VW(#SET_TIME,TRUE,11,1,0)
      ;ENDFOLD
      ;FOLD -- ServoGun SZ1 schliessen -- ;%{SE}%MKUKATPVW %CVW_COM %VCOMMENT %P 2:-- ServoGun SZ1 schliessen --, 3: VW_COMMENT
      ;ENDFOLD
      ;FOLD A3935 = !E1156 & E1157 & E1158 & !E1159 ;%{SE}%MKUKATPVW %CVW_SPS %VBOASG %P 2:A3935 = !E1156 & E1157 & E1158 & !E1159, 3: BOASG
         $OUT[3935] = NOT $IN[1156] AND $IN[1157] AND $IN[1158] AND NOT $IN[1159]
      ;ENDFOLD
      ;FOLD -- KF1 Ausblasen -- ;%{SE}%MKUKATPVW %CVW_COM %VCOMMENT %P 2:-- KF1 Ausblasen --, 3: VW_COMMENT
      ;ENDFOLD
      ;FOLD A1156 = F330 + F331 + !F330 & !F331 & !F332 ;%{SE}%MKUKATPVW %CVW_SPS %VBOASG %P 2:A1156 = F330 + F331 + !F330 & !F331 & !F332, 3: BOASG
         $OUT[1156] = $FLAG[330] OR $FLAG[331] OR NOT $FLAG[330] AND NOT $FLAG[331] AND NOT $FLAG[332]
      ;ENDFOLD
      ;FOLD SCHRITT 314 = !A3926 & A3928 & A4039 + T9 ;%{SE}%MKUKATPVW %CVW_SPS %VST_CON %P 2:SCHRITT 314 = !A3926 & A3928 & A4039 + T9, 3: ST_CON
         IF NOT $OUT[3926] AND $OUT[3928] AND $OUT[4039] OR $TIMER_FLAG[9] THEN
            PREV_STEP[9] = APP_INT_STEP[9]
            APP_INT_STEP[9] = 314
         ENDIF
      ;ENDFOLD
   ;ENDFOLD
   ;FOLD SCHRITT 314 -- st. RZ3 -- ;%{P}%MKUKATPVW,%CSTEP,%VST_NR,%P 1:SCHRITT, 2:314, 3: st. RZ3
      ;FOLD ;%{H}
         Case 314
      ;ENDFOLD
      ;FOLD -- RSK Fehlerausgabe Kraftaufbau -- ;%{SE}%MKUKATPVW %CVW_COM %VCOMMENT %P 2:-- RSK Fehlerausgabe Kraftaufbau --, 3: VW_COMMENT
      ;ENDFOLD
      ;FOLD F325 = T9 ;%{SE}%MKUKATPVW %CVW_SPS %VBOASG %P 2:F325 = T9, 3: BOASG
         $FLAG[325] = $TIMER_FLAG[9]
      ;ENDFOLD
      ;FOLD -- RSK Sammelstoerung -- ;%{SE}%MKUKATPVW %CVW_COM %VCOMMENT %P 2:-- RSK Sammelstoerung --, 3: VW_COMMENT
      ;ENDFOLD
      ;FOLD F329 = F325 ;%{SE}%MKUKATPVW %CVW_SPS %VBOASG %P 2:F329 = F325, 3: BOASG
         $FLAG[329] = $FLAG[325]
      ;ENDFOLD
      ;FOLD -- KF1 abschalten bei Fehler -- ;%{SE}%MKUKATPVW %CVW_COM %VCOMMENT %P 2:-- KF1 abschalten bei Fehler --, 3: VW_COMMENT
      ;ENDFOLD
      ;FOLD A1154 = !T9 ;%{SE}%MKUKATPVW %CVW_SPS %VBOASG %P 2:A1154 = !T9, 3: BOASG
         $OUT[1154] = NOT $TIMER_FLAG[9]
      ;ENDFOLD
      ;FOLD -- KF1 Ausblasen -- ;%{SE}%MKUKATPVW %CVW_COM %VCOMMENT %P 2:-- KF1 Ausblasen --, 3: VW_COMMENT
      ;ENDFOLD
      ;FOLD A1156 = (F330 + F331 + !F330 & !F331 & !F332) & !T9 ;%{SE}%MKUKATPVW %CVW_SPS %VBOASG %P 2:A1156 = (F330 + F331 + !F330 & !F331 & !F332) & !T9, 3: BOASG
         $OUT[1156] = ($FLAG[330] OR $FLAG[331] OR NOT $FLAG[330] AND NOT $FLAG[331] AND NOT $FLAG[332]) AND NOT $TIMER_FLAG[9]
      ;ENDFOLD
      ;FOLD -- Warte Fraesen fertig oder Timeout -- ;%{SE}%MKUKATPVW %CVW_COM %VCOMMENT %P 2:-- Warte Fraesen fertig oder Timeout --, 3: VW_COMMENT
      ;ENDFOLD
      ;FOLD SCHRITT 315 = (F175 & F190 + F174 & F186 & !F287 + T7 + T9 + F325) & A4039 ;%{SE}%MKUKATPVW %CVW_SPS %VST_CON %P 2:SCHRITT 315 = (F175 & F190 + F174 & F186 & !F287 + T7 + T9 + F325) & A4039, 3: ST_CON
         IF ($FLAG[175] AND $FLAG[190] OR $FLAG[174] AND $FLAG[186] AND NOT $FLAG[287] OR $TIMER_FLAG[7] OR $TIMER_FLAG[9] OR $FLAG[325]) AND $OUT[4039] THEN
            PREV_STEP[9] = APP_INT_STEP[9]
            APP_INT_STEP[9] = 315
         ENDIF
      ;ENDFOLD
      ;FOLD SCHRITT 315 = (F174 & F188 & F287 + T7 + T9 + F325) & A4039 ;%{SE}%MKUKATPVW %CVW_SPS %VST_CON %P 2:SCHRITT 315 = (F174 & F188 & F287 + T7 + T9 + F325) & A4039, 3: ST_CON
         IF ($FLAG[174] AND $FLAG[188] AND $FLAG[287] OR $TIMER_FLAG[7] OR $TIMER_FLAG[9] OR $FLAG[325]) AND $OUT[4039] THEN
            PREV_STEP[9] = APP_INT_STEP[9]
            APP_INT_STEP[9] = 315
         ENDIF
      ;ENDFOLD
   ;ENDFOLD
   ;FOLD SCHRITT 315 -- st. RZ3 # GunOpen -- ;%{P}%MKUKATPVW,%CSTEP,%VST_NR,%P 1:SCHRITT, 2:315, 3: st. RZ3 # GunOpen
      ;FOLD ;%{H}
         Case 315
      ;ENDFOLD
      ;FOLD -- ServoGun SZ1 oeffnen -- ;%{SE}%MKUKATPVW %CVW_COM %VCOMMENT %P 2:-- ServoGun SZ1 oeffnen --, 3: VW_COMMENT
      ;ENDFOLD
      ;FOLD t9 ( EIN ) = STOP ;%{SE}%MKUKATPVW %CVW_SPS %VTSTOP %P 2:t9 ( EIN ) = STOP, 3: TSTOP
         VW(#SET_TIME,TRUE,9,1,0)
      ;ENDFOLD
      ;FOLD A3935 = AUS ;%{SE}%MKUKATPVW %CVW_SPS %VBOASG %P 2:A3935 = AUS, 3: BOASG
         $OUT[3935] = FALSE
      ;ENDFOLD
      ;FOLD A3936 = EIN ;%{SE}%MKUKATPVW %CVW_SPS %VBOASG %P 2:A3936 = EIN, 3: BOASG
         $OUT[3936] = TRUE
      ;ENDFOLD
      ;FOLD -- KF1 Ausblasen -- ;%{SE}%MKUKATPVW %CVW_COM %VCOMMENT %P 2:-- KF1 Ausblasen --, 3: VW_COMMENT
      ;ENDFOLD
      ;FOLD A1156 = (F330 + F331 + F332 + !F330 & !F331 & !F332) & !T9 ;%{SE}%MKUKATPVW %CVW_SPS %VBOASG %P 2:A1156 = (F330 + F331 + F332 + !F330 & !F331 & !F332) & !T9, 3: BOASG
         $OUT[1156] = ($FLAG[330] OR $FLAG[331] OR $FLAG[332] OR NOT $FLAG[330] AND NOT $FLAG[331] AND NOT $FLAG[332]) AND NOT $TIMER_FLAG[9]
      ;ENDFOLD
      ;FOLD -- KF Ausblasen Ausschaltverzoegerung starten -- ;%{SE}%MKUKATPVW %CVW_COM %VCOMMENT %P 2:-- KF Ausblasen Ausschaltverzoegerung starten --, 3: VW_COMMENT
      ;ENDFOLD
      ;FOLD F737 = AUS ;%{SE}%MKUKATPVW %CVW_SPS %VBOASG %P 2:F737 = AUS, 3: BOASG
         $FLAG[737] = FALSE
      ;ENDFOLD
      ;FOLD -- RSK Sammelstoerung -- ;%{SE}%MKUKATPVW %CVW_COM %VCOMMENT %P 2:-- RSK Sammelstoerung --, 3: VW_COMMENT
      ;ENDFOLD
      ;FOLD F329 = T7 + T9 + F325 ;%{SE}%MKUKATPVW %CVW_SPS %VBOASG %P 2:F329 = T7 + T9 + F325, 3: BOASG
         $FLAG[329] = $TIMER_FLAG[7] OR $TIMER_FLAG[9] OR $FLAG[325]
      ;ENDFOLD
      ;FOLD -- Hilfsflag Startfraesen -- ;%{SE}%MKUKATPVW %CVW_COM %VCOMMENT %P 2:-- Hilfsflag Startfraesen --, 3: VW_COMMENT
      ;ENDFOLD
      ;FOLD F188 = F188 & F287 ;%{SE}%MKUKATPVW %CVW_SPS %VBOASG %P 2:F188 = F188 & F287, 3: BOASG
         $FLAG[188] = $FLAG[188] AND $FLAG[287]
      ;ENDFOLD
      ;FOLD F188 = (F188 & F174 + F190 & F175) & F287 ;%{SE}%MKUKATPVW %CVW_SPS %VBOASG %P 2:F188 = (F188 & F174 + F190 & F175) & F287, 3: BOASG
         $FLAG[188] = ($FLAG[188] AND $FLAG[174] OR $FLAG[190] AND $FLAG[175]) AND $FLAG[287]
      ;ENDFOLD
      ;FOLD F190 = !F130 & F190 + F130 & F287 & F190 ;%{SE}%MKUKATPVW %CVW_SPS %VBOASG %P 2:F190 = !F130 & F190 + F130 & F287 & F190, 3: BOASG
         $FLAG[190] = NOT $FLAG[130] AND $FLAG[190] OR $FLAG[130] AND $FLAG[287] AND $FLAG[190]
      ;ENDFOLD
      ;FOLD F287 = F174 + F175 & F130 ;%{SE}%MKUKATPVW %CVW_SPS %VBOASG %P 2:F287 = F174 + F175 & F130, 3: BOASG
         $FLAG[287] = $FLAG[174] OR $FLAG[175] AND $FLAG[130]
      ;ENDFOLD
      ;FOLD -- Neues Fraesprogramm und Zaehler ruecksetzen -- ;%{SE}%MKUKATPVW %CVW_COM %VCOMMENT %P 2:-- Neues Fraesprogramm und Zaehler ruecksetzen --, 3: VW_COMMENT
      ;ENDFOLD
      ;FOLD bin31 ( F200 ) = 36 ;%{SE}%MKUKATPVW %CVW_SPS %VARIASG %P 2:bin31 ( F200 ) = 36, 3: ARIASG
         VW(#BINOUT,$FLAG[200],31,36)
      ;ENDFOLD
      ;FOLD i19 ( F188 ) = i45 ;%{SE}%MKUKATPVW %CVW_SPS %VARIASG %P 2:i19 ( F188 ) = i45, 3: ARIASG
         VW(#COUNTER,$FLAG[188],19,$COUNT_I[45])
      ;ENDFOLD
      ;FOLD -- Wiederholung beim Startfraesen -- ;%{SE}%MKUKATPVW %CVW_COM %VCOMMENT %P 2:-- Wiederholung beim Startfraesen --, 3: VW_COMMENT
      ;ENDFOLD
      ;FOLD SCHRITT 311 = A3926 & A3508 & (F174 & !F188 + F175 & F130 & !F188) & !F329 & A4039 & A3520 ;%{SE}%MKUKATPVW %CVW_SPS %VST_CON %P 2:SCHRITT 311 = A3926 & A3508 & (F174 & !F188 + F175 & F130 & !F188) & !F329 & A4039 & A3520, 3: ST_CON
         IF $OUT[3926] AND $OUT[3508] AND ($FLAG[174] AND NOT $FLAG[188] OR $FLAG[175] AND $FLAG[130] AND NOT $FLAG[188]) AND NOT $FLAG[329] AND $OUT[4039] AND $OUT[3520] THEN
            PREV_STEP[9] = APP_INT_STEP[9]
            APP_INT_STEP[9] = 311
         ENDIF
      ;ENDFOLD
      ;FOLD -- Wiederholung beim Startfraesen -- ;%{SE}%MKUKATPVW %CVW_COM %VCOMMENT %P 2:-- Wiederholung beim Startfraesen --, 3: VW_COMMENT
      ;ENDFOLD
      ;FOLD SCHRITT 316 = A3926 & A3508 & (F174 & !F188 + F175 & F130 & !F188) & !F329 & A4039 & !A3520 ;%{SE}%MKUKATPVW %CVW_SPS %VST_CON %P 2:SCHRITT 316 = A3926 & A3508 & (F174 & !F188 + F175 & F130 & !F188) & !F329 & A4039 & !A3520, 3: ST_CON
         IF $OUT[3926] AND $OUT[3508] AND ($FLAG[174] AND NOT $FLAG[188] OR $FLAG[175] AND $FLAG[130] AND NOT $FLAG[188]) AND NOT $FLAG[329] AND $OUT[4039] AND NOT $OUT[3520] THEN
            PREV_STEP[9] = APP_INT_STEP[9]
            APP_INT_STEP[9] = 316
         ENDIF
      ;ENDFOLD
      ;FOLD -- Weiter wenn Fraesen fertig -- ;%{SE}%MKUKATPVW %CVW_COM %VCOMMENT %P 2:-- Weiter wenn Fraesen fertig --, 3: VW_COMMENT
      ;ENDFOLD
      ;FOLD SCHRITT 316 = A3926 & A3508 & (F175 & F190 & (!F130 + F188) + F174 & F188 + F329 + F325) & A4039 ;%{SE}%MKUKATPVW %CVW_SPS %VST_CON %P 2:SCHRITT 316 = A3926 & A3508 & (F175 & F190 & (!F130 + F188) + F174 & F188 + F329 + F325) & A4039, 3: ST_CON
         IF $OUT[3926] AND $OUT[3508] AND ($FLAG[175] AND $FLAG[190] AND (NOT $FLAG[130] OR $FLAG[188]) OR $FLAG[174] AND $FLAG[188] OR $FLAG[329] OR $FLAG[325]) AND $OUT[4039] THEN
            PREV_STEP[9] = APP_INT_STEP[9]
            APP_INT_STEP[9] = 316
         ENDIF
      ;ENDFOLD
   ;ENDFOLD
   ;FOLD SCHRITT 316 -- st. RZ3 # Acknowledge -- ;%{P}%MKUKATPVW,%CSTEP,%VST_NR,%P 1:SCHRITT, 2:316, 3: st. RZ3 # Acknowledge
      ;FOLD ;%{H}
         Case 316
      ;ENDFOLD
      ;FOLD -- Hilfsflag Durchlaufmerker -- ;%{SE}%MKUKATPVW %CVW_COM %VCOMMENT %P 2:-- Hilfsflag Durchlaufmerker --, 3: VW_COMMENT
      ;ENDFOLD
      ;FOLD F324 = AUS ;%{SE}%MKUKATPVW %CVW_SPS %VBOASG %P 2:F324 = AUS, 3: BOASG
         $FLAG[324] = FALSE
      ;ENDFOLD
      ;FOLD A3935 = AUS ;%{SE}%MKUKATPVW %CVW_SPS %VBOASG %P 2:A3935 = AUS, 3: BOASG
         $OUT[3935] = FALSE
      ;ENDFOLD
      ;FOLD A3936 = AUS ;%{SE}%MKUKATPVW %CVW_SPS %VBOASG %P 2:A3936 = AUS, 3: BOASG
         $OUT[3936] = FALSE
      ;ENDFOLD
      ;FOLD A3510 = AUS ;%{SE}%MKUKATPVW %CVW_SPS %VBOASG %P 2:A3510 = AUS, 3: BOASG
         $OUT[3510] = FALSE
      ;ENDFOLD
      ;FOLD A3512 = EIN ;%{SE}%MKUKATPVW %CVW_SPS %VBOASG %P 2:A3512 = EIN, 3: BOASG
         $OUT[3512] = TRUE
      ;ENDFOLD
      ;FOLD t9 ( EIN ) = STOP ;%{SE}%MKUKATPVW %CVW_SPS %VTSTOP %P 2:t9 ( EIN ) = STOP, 3: TSTOP
         VW(#SET_TIME,TRUE,9,1,0)
      ;ENDFOLD
      ;FOLD -- KF1 abschalten -- ;%{SE}%MKUKATPVW %CVW_COM %VCOMMENT %P 2:-- KF1 abschalten --, 3: VW_COMMENT
      ;ENDFOLD
      ;FOLD A1154 = AUS ;%{SE}%MKUKATPVW %CVW_SPS %VBOASG %P 2:A1154 = AUS, 3: BOASG
         $OUT[1154] = FALSE
      ;ENDFOLD
      ;FOLD -- Ueberwachungszeit KF1 Versetzeinheit -- ;%{SE}%MKUKATPVW %CVW_COM %VCOMMENT %P 2:-- Ueberwachungszeit KF1 Versetzeinheit --, 3: VW_COMMENT
      ;ENDFOLD
      ;FOLD t8 ( EIN ) = -40[1/10Sek] ;%{SE}%MKUKATPVW %CVW_SPS %VTASG %P 2:t8 ( EIN ) = -40[1/10Sek], 3: TASG
         VW(#SET_TIME,TRUE,8,0,-40)
      ;ENDFOLD
      ;FOLD SCHRITT 317 = A4039 & !E195 ;%{SE}%MKUKATPVW %CVW_SPS %VST_CON %P 2:SCHRITT 317 = A4039 & !E195, 3: ST_CON
         IF $OUT[4039] AND NOT $IN[195] THEN
            PREV_STEP[9] = APP_INT_STEP[9]
            APP_INT_STEP[9] = 317
         ENDIF
      ;ENDFOLD
   ;ENDFOLD
   ;FOLD SCHRITT 317 -- st. RZ3 -- ;%{P}%MKUKATPVW,%CSTEP,%VST_NR,%P 1:SCHRITT, 2:317, 3: st. RZ3
      ;FOLD ;%{H}
         Case 317
      ;ENDFOLD
      ;FOLD -- RSK Fehlerausgabe Arbeitsst. -- ;%{SE}%MKUKATPVW %CVW_COM %VCOMMENT %P 2:-- RSK Fehlerausgabe Arbeitsst. --, 3: VW_COMMENT
      ;ENDFOLD
      ;FOLD F328 = AUS ;%{SE}%MKUKATPVW %CVW_SPS %VBOASG %P 2:F328 = AUS, 3: BOASG
         $FLAG[328] = FALSE
      ;ENDFOLD
      ;FOLD -- KF1 Versetzeinheit vor -- ;%{SE}%MKUKATPVW %CVW_COM %VCOMMENT %P 2:-- KF1 Versetzeinheit vor --, 3: VW_COMMENT
      ;ENDFOLD
      ;FOLD A1155 = F564 ;%{SE}%MKUKATPVW %CVW_SPS %VBOASG %P 2:A1155 = F564, 3: BOASG
         $OUT[1155] = $FLAG[564]
      ;ENDFOLD
      ;FOLD A3512 = AUS ;%{SE}%MKUKATPVW %CVW_SPS %VBOASG %P 2:A3512 = AUS, 3: BOASG
         $OUT[3512] = FALSE
      ;ENDFOLD
      ;FOLD -- RSK Fehlerausgabe KS1 Arbeitsst. -- ;%{SE}%MKUKATPVW %CVW_COM %VCOMMENT %P 2:-- RSK Fehlerausgabe KS1 Arbeitsst. --, 3: VW_COMMENT
      ;ENDFOLD
      ;FOLD F324 = (E1156 + !E1157 + !E1158 + E1159) & !F323 & !F328 + F324 ;%{SE}%MKUKATPVW %CVW_SPS %VBOASG %P 2:F324 = (E1156 + !E1157 + !E1158 + E1159) & !F323 & !F328 + F324, 3: BOASG
         $FLAG[324] = ($IN[1156] OR NOT $IN[1157] OR NOT $IN[1158] OR $IN[1159]) AND NOT $FLAG[323] AND NOT $FLAG[328] OR $FLAG[324]
      ;ENDFOLD
      ;FOLD -- RSK Sammelstoerung -- ;%{SE}%MKUKATPVW %CVW_COM %VCOMMENT %P 2:-- RSK Sammelstoerung --, 3: VW_COMMENT
      ;ENDFOLD
      ;FOLD F329 = F324 + F325 ;%{SE}%MKUKATPVW %CVW_SPS %VBOASG %P 2:F329 = F324 + F325, 3: BOASG
         $FLAG[329] = $FLAG[324] OR $FLAG[325]
      ;ENDFOLD
      ;FOLD -- Ueberwachungszeit KS1 schwenken -- ;%{SE}%MKUKATPVW %CVW_COM %VCOMMENT %P 2:-- Ueberwachungszeit KS1 schwenken --, 3: VW_COMMENT
      ;ENDFOLD
      ;FOLD t9 ( EIN ) = -100[1/10Sek] ;%{SE}%MKUKATPVW %CVW_SPS %VTASG %P 2:t9 ( EIN ) = -100[1/10Sek], 3: TASG
         VW(#SET_TIME,TRUE,9,0,-100)
      ;ENDFOLD
      ;FOLD SCHRITT 316 = F324 & (E26 + E27) & A4039 ;%{SE}%MKUKATPVW %CVW_SPS %VST_CON %P 2:SCHRITT 316 = F324 & (E26 + E27) & A4039, 3: ST_CON
         IF $FLAG[324] AND ($IN[26] OR $IN[27]) AND $OUT[4039] THEN
            PREV_STEP[9] = APP_INT_STEP[9]
            APP_INT_STEP[9] = 316
         ENDIF
      ;ENDFOLD
      ;FOLD SCHRITT 318 = (!F324 & (E1155 & F564 + !E1155 & !F564) + T8 + F325) & A4039 ;%{SE}%MKUKATPVW %CVW_SPS %VST_CON %P 2:SCHRITT 318 = (!F324 & (E1155 & F564 + !E1155 & !F564) + T8 + F325) & A4039, 3: ST_CON
         IF (NOT $FLAG[324] AND ($IN[1155] AND $FLAG[564] OR NOT $IN[1155] AND NOT $FLAG[564]) OR $TIMER_FLAG[8] OR $FLAG[325]) AND $OUT[4039] THEN
            PREV_STEP[9] = APP_INT_STEP[9]
            APP_INT_STEP[9] = 318
         ENDIF
      ;ENDFOLD
   ;ENDFOLD
   ;FOLD SCHRITT 318 -- st. RZ3 -- ;%{P}%MKUKATPVW,%CSTEP,%VST_NR,%P 1:SCHRITT, 2:318, 3: st. RZ3
      ;FOLD ;%{H}
         Case 318
      ;ENDFOLD
      ;FOLD F323 = AUS ;%{SE}%MKUKATPVW %CVW_SPS %VBOASG %P 2:F323 = AUS, 3: BOASG
         $FLAG[323] = FALSE
      ;ENDFOLD
      ;FOLD F328 = AUS ;%{SE}%MKUKATPVW %CVW_SPS %VBOASG %P 2:F328 = AUS, 3: BOASG
         $FLAG[328] = FALSE
      ;ENDFOLD
      ;FOLD -- RSK Sammelstoerung -- ;%{SE}%MKUKATPVW %CVW_COM %VCOMMENT %P 2:-- RSK Sammelstoerung --, 3: VW_COMMENT
      ;ENDFOLD
      ;FOLD F329 = F325 ;%{SE}%MKUKATPVW %CVW_SPS %VBOASG %P 2:F329 = F325, 3: BOASG
         $FLAG[329] = $FLAG[325]
      ;ENDFOLD
      ;FOLD -- KF1 ein -- ;%{SE}%MKUKATPVW %CVW_COM %VCOMMENT %P 2:-- KF1 ein --, 3: VW_COMMENT
      ;ENDFOLD
      ;FOLD A1154 = EIN ;%{SE}%MKUKATPVW %CVW_SPS %VBOASG %P 2:A1154 = EIN, 3: BOASG
         $OUT[1154] = TRUE
      ;ENDFOLD
      ;FOLD -- KF Ausblasen Ausschaltverzoegerung starten -- ;%{SE}%MKUKATPVW %CVW_COM %VCOMMENT %P 2:-- KF Ausblasen Ausschaltverzoegerung starten --, 3: VW_COMMENT
      ;ENDFOLD
      ;FOLD F737 = EIN ;%{SE}%MKUKATPVW %CVW_SPS %VBOASG %P 2:F737 = EIN, 3: BOASG
         $FLAG[737] = TRUE
      ;ENDFOLD
      ;FOLD -- KF1 Ausblasen -- ;%{SE}%MKUKATPVW %CVW_COM %VCOMMENT %P 2:-- KF1 Ausblasen --, 3: VW_COMMENT
      ;ENDFOLD
      ;FOLD A1156 = (F330 + F331 + F332) & F737 ;%{SE}%MKUKATPVW %CVW_SPS %VBOASG %P 2:A1156 = (F330 + F331 + F332) & F737, 3: BOASG
         $OUT[1156] = ($FLAG[330] OR $FLAG[331] OR $FLAG[332]) AND $FLAG[737]
      ;ENDFOLD
      ;FOLD -- KS1 in Ruhestellung schwenken -- ;%{SE}%MKUKATPVW %CVW_COM %VCOMMENT %P 2:-- KS1 in Ruhestellung schwenken --, 3: VW_COMMENT
      ;ENDFOLD
      ;FOLD A1160 = A3862 & (E1155 & F564 + !E1155 & !F564) ;%{SE}%MKUKATPVW %CVW_SPS %VBOASG %P 2:A1160 = A3862 & (E1155 & F564 + !E1155 & !F564), 3: BOASG
         $OUT[1160] = $OUT[3862] AND ($IN[1155] AND $FLAG[564] OR NOT $IN[1155] AND NOT $FLAG[564])
      ;ENDFOLD
      ;FOLD SCHRITT 320 = A3926 & A1160 & A4039 + T9 ;%{SE}%MKUKATPVW %CVW_SPS %VST_CON %P 2:SCHRITT 320 = A3926 & A1160 & A4039 + T9, 3: ST_CON
         IF $OUT[3926] AND $OUT[1160] AND $OUT[4039] OR $TIMER_FLAG[9] THEN
            PREV_STEP[9] = APP_INT_STEP[9]
            APP_INT_STEP[9] = 320
         ENDIF
      ;ENDFOLD
   ;ENDFOLD
   ;FOLD SCHRITT 320 -- st. RZ3 -- ;%{P}%MKUKATPVW,%CSTEP,%VST_NR,%P 1:SCHRITT, 2:320, 3: st. RZ3
      ;FOLD ;%{H}
         Case 320
      ;ENDFOLD
      ;FOLD -- Hilfsflag SK Programmwechsel -- ;%{SE}%MKUKATPVW %CVW_COM %VCOMMENT %P 2:-- Hilfsflag SK Programmwechsel --, 3: VW_COMMENT
      ;ENDFOLD
      ;FOLD F334 = AUS ;%{SE}%MKUKATPVW %CVW_SPS %VBOASG %P 2:F334 = AUS, 3: BOASG
         $FLAG[334] = FALSE
      ;ENDFOLD
      ;FOLD -- RSK Fehlerausgabe KF Versetzeinheit -- ;%{SE}%MKUKATPVW %CVW_COM %VCOMMENT %P 2:-- RSK Fehlerausgabe KF Versetzeinheit --, 3: VW_COMMENT
      ;ENDFOLD
      ;FOLD F328 = !E1155 & F564 & !F323 + F328 ;%{SE}%MKUKATPVW %CVW_SPS %VBOASG %P 2:F328 = !E1155 & F564 & !F323 + F328, 3: BOASG
         $FLAG[328] = NOT $IN[1155] AND $FLAG[564] AND NOT $FLAG[323] OR $FLAG[328]
      ;ENDFOLD
      ;FOLD -- RSK Fehlerausgabe KS1 Ruhestellung -- ;%{SE}%MKUKATPVW %CVW_COM %VCOMMENT %P 2:-- RSK Fehlerausgabe KS1 Ruhestellung --, 3: VW_COMMENT
      ;ENDFOLD
      ;FOLD F323 = (!E1156 + E1157 + E1158 + !E1159) & T9 & (E1155 + !F564) + F323 ;%{SE}%MKUKATPVW %CVW_SPS %VBOASG %P 2:F323 = (!E1156 + E1157 + E1158 + !E1159) & T9 & (E1155 + !F564) + F323, 3: BOASG
         $FLAG[323] = (NOT $IN[1156] OR $IN[1157] OR $IN[1158] OR NOT $IN[1159]) AND $TIMER_FLAG[9] AND ($IN[1155] OR NOT $FLAG[564]) OR $FLAG[323]
      ;ENDFOLD
      ;FOLD -- RSK Fehlerausgabe EZ/SP min. Oeffnung -- ;%{SE}%MKUKATPVW %CVW_COM %VCOMMENT %P 2:-- RSK Fehlerausgabe EZ/SP min. Oeffnung --, 3: VW_COMMENT
      ;ENDFOLD
      ;FOLD F333 = !A3926 ;%{SE}%MKUKATPVW %CVW_SPS %VBOASG %P 2:F333 = !A3926, 3: BOASG
         $FLAG[333] = NOT $OUT[3926]
      ;ENDFOLD
      ;FOLD -- RSK Sammelstoerung -- ;%{SE}%MKUKATPVW %CVW_COM %VCOMMENT %P 2:-- RSK Sammelstoerung --, 3: VW_COMMENT
      ;ENDFOLD
      ;FOLD F329 = F323 + F325 + F328 + F333 ;%{SE}%MKUKATPVW %CVW_SPS %VBOASG %P 2:F329 = F323 + F325 + F328 + F333, 3: BOASG
         $FLAG[329] = $FLAG[323] OR $FLAG[325] OR $FLAG[328] OR $FLAG[333]
      ;ENDFOLD
      ;FOLD A1154 = !F323 & !F328 ;%{SE}%MKUKATPVW %CVW_SPS %VBOASG %P 2:A1154 = !F323 & !F328, 3: BOASG
         $OUT[1154] = NOT $FLAG[323] AND NOT $FLAG[328]
      ;ENDFOLD
      ;FOLD A1155 = F564 ;%{SE}%MKUKATPVW %CVW_SPS %VBOASG %P 2:A1155 = F564, 3: BOASG
         $OUT[1155] = $FLAG[564]
      ;ENDFOLD
      ;FOLD SCHRITT 316 = (F323 + F328) & (E26 + E27) & A4039 ;%{SE}%MKUKATPVW %CVW_SPS %VST_CON %P 2:SCHRITT 316 = (F323 + F328) & (E26 + E27) & A4039, 3: ST_CON
         IF ($FLAG[323] OR $FLAG[328]) AND ($IN[26] OR $IN[27]) AND $OUT[4039] THEN
            PREV_STEP[9] = APP_INT_STEP[9]
            APP_INT_STEP[9] = 316
         ENDIF
      ;ENDFOLD
      ;FOLD SCHRITT 321 = !A1160 & E1156 & !E1157 & !E1158 & E1159 & A4039 ;%{SE}%MKUKATPVW %CVW_SPS %VST_CON %P 2:SCHRITT 321 = !A1160 & E1156 & !E1157 & !E1158 & E1159 & A4039, 3: ST_CON
         IF NOT $OUT[1160] AND $IN[1156] AND NOT $IN[1157] AND NOT $IN[1158] AND $IN[1159] AND $OUT[4039] THEN
            PREV_STEP[9] = APP_INT_STEP[9]
            APP_INT_STEP[9] = 321
         ENDIF
      ;ENDFOLD
   ;ENDFOLD
   ;FOLD SCHRITT 321 -- st. RZ3 -- ;%{P}%MKUKATPVW,%CSTEP,%VST_NR,%P 1:SCHRITT, 2:321, 3: st. RZ3
      ;FOLD ;%{H}
         Case 321
      ;ENDFOLD
      ;FOLD F323 = AUS ;%{SE}%MKUKATPVW %CVW_SPS %VBOASG %P 2:F323 = AUS, 3: BOASG
         $FLAG[323] = FALSE
      ;ENDFOLD
      ;FOLD F328 = AUS ;%{SE}%MKUKATPVW %CVW_SPS %VBOASG %P 2:F328 = AUS, 3: BOASG
         $FLAG[328] = FALSE
      ;ENDFOLD
      ;FOLD -- KF Ausblasen Ausschaltverzoegerung starten -- ;%{SE}%MKUKATPVW %CVW_COM %VCOMMENT %P 2:-- KF Ausblasen Ausschaltverzoegerung starten --, 3: VW_COMMENT
      ;ENDFOLD
      ;FOLD F737 = EIN ;%{SE}%MKUKATPVW %CVW_SPS %VBOASG %P 2:F737 = EIN, 3: BOASG
         $FLAG[737] = TRUE
      ;ENDFOLD
      ;FOLD -- RSK Sammelstoerung -- ;%{SE}%MKUKATPVW %CVW_COM %VCOMMENT %P 2:-- RSK Sammelstoerung --, 3: VW_COMMENT
      ;ENDFOLD
      ;FOLD F329 = F325 ;%{SE}%MKUKATPVW %CVW_SPS %VBOASG %P 2:F329 = F325, 3: BOASG
         $FLAG[329] = $FLAG[325]
      ;ENDFOLD
      ;FOLD t9 ( EIN ) = STOP ;%{SE}%MKUKATPVW %CVW_SPS %VTSTOP %P 2:t9 ( EIN ) = STOP, 3: TSTOP
         VW(#SET_TIME,TRUE,9,1,0)
      ;ENDFOLD
      ;FOLD -- KF1 Versetzeinheit rueck -- ;%{SE}%MKUKATPVW %CVW_COM %VCOMMENT %P 2:-- KF1 Versetzeinheit rueck --, 3: VW_COMMENT
      ;ENDFOLD
      ;FOLD A1155 = AUS ;%{SE}%MKUKATPVW %CVW_SPS %VBOASG %P 2:A1155 = AUS, 3: BOASG
         $OUT[1155] = FALSE
      ;ENDFOLD
      ;FOLD -- KF1 aus -- ;%{SE}%MKUKATPVW %CVW_COM %VCOMMENT %P 2:-- KF1 aus --, 3: VW_COMMENT
      ;ENDFOLD
      ;FOLD A1154 = AUS ;%{SE}%MKUKATPVW %CVW_SPS %VBOASG %P 2:A1154 = AUS, 3: BOASG
         $OUT[1154] = FALSE
      ;ENDFOLD
      ;FOLD -- KF1 Ausblasen -- ;%{SE}%MKUKATPVW %CVW_COM %VCOMMENT %P 2:-- KF1 Ausblasen --, 3: VW_COMMENT
      ;ENDFOLD
      ;FOLD A1156 = (F330 + F331 + F332) & F737 ;%{SE}%MKUKATPVW %CVW_SPS %VBOASG %P 2:A1156 = (F330 + F331 + F332) & F737, 3: BOASG
         $OUT[1156] = ($FLAG[330] OR $FLAG[331] OR $FLAG[332]) AND $FLAG[737]
      ;ENDFOLD
      ;FOLD bin7 ( !F329 ) = 1 ;%{SE}%MKUKATPVW %CVW_SPS %VARIASG %P 2:bin7 ( !F329 ) = 1, 3: ARIASG
         VW(#BINOUT,NOT $FLAG[329],7,1)
      ;ENDFOLD
      ;FOLD bin9 ( !F329 ) = 1 ;%{SE}%MKUKATPVW %CVW_SPS %VARIASG %P 2:bin9 ( !F329 ) = 1, 3: ARIASG
         VW(#BINOUT,NOT $FLAG[329],9,1)
      ;ENDFOLD
      ;FOLD bin31 ( !F329 ) = 1 ;%{SE}%MKUKATPVW %CVW_SPS %VARIASG %P 2:bin31 ( !F329 ) = 1, 3: ARIASG
         VW(#BINOUT,NOT $FLAG[329],31,1)
      ;ENDFOLD
      ;FOLD -- Wartezeit Programmwechsel SK -- ;%{SE}%MKUKATPVW %CVW_COM %VCOMMENT %P 2:-- Wartezeit Programmwechsel SK --, 3: VW_COMMENT
      ;ENDFOLD
      ;FOLD T8 ( !F334 ) = -2[1/10Sek] ;%{SE}%MKUKATPVW %CVW_SPS %VTASG %P 2:T8 ( !F334 ) = -2[1/10Sek], 3: TASG
         VW(#SET_TIME,NOT $FLAG[334],8,0,-2)
      ;ENDFOLD
      ;FOLD -- Hilfsflag SK Programmwechsel -- ;%{SE}%MKUKATPVW %CVW_COM %VCOMMENT %P 2:-- Hilfsflag SK Programmwechsel --, 3: VW_COMMENT
      ;ENDFOLD
      ;FOLD F334 = EIN ;%{SE}%MKUKATPVW %CVW_SPS %VBOASG %P 2:F334 = EIN, 3: BOASG
         $FLAG[334] = TRUE
      ;ENDFOLD
      ;FOLD SCHRITT 303 = (F325 + F329) & (E26 + E27) & A4039 ;%{SE}%MKUKATPVW %CVW_SPS %VST_CON %P 2:SCHRITT 303 = (F325 + F329) & (E26 + E27) & A4039, 3: ST_CON
         IF ($FLAG[325] OR $FLAG[329]) AND ($IN[26] OR $IN[27]) AND $OUT[4039] THEN
            PREV_STEP[9] = APP_INT_STEP[9]
            APP_INT_STEP[9] = 303
         ENDIF
      ;ENDFOLD
      ;FOLD SCHRITT 322 = T8 & !F325 & !F329 & A4039 & (A3506 & A3505) ;%{SE}%MKUKATPVW %CVW_SPS %VST_CON %P 2:SCHRITT 322 = T8 & !F325 & !F329 & A4039 & (A3506 & A3505), 3: ST_CON
         IF $TIMER_FLAG[8] AND NOT $FLAG[325] AND NOT $FLAG[329] AND $OUT[4039] AND ($OUT[3506] AND $OUT[3505]) THEN
            PREV_STEP[9] = APP_INT_STEP[9]
            APP_INT_STEP[9] = 322
         ENDIF
      ;ENDFOLD
   ;ENDFOLD
   ;FOLD SCHRITT 322 -- st. RZ3 -- ;%{P}%MKUKATPVW,%CSTEP,%VST_NR,%P 1:SCHRITT, 2:322, 3: st. RZ3
      ;FOLD ;%{H}
         Case 322
      ;ENDFOLD
      ;FOLD -- Hilfsflag SK Programmwechsel -- ;%{SE}%MKUKATPVW %CVW_COM %VCOMMENT %P 2:-- Hilfsflag SK Programmwechsel --, 3: VW_COMMENT
      ;ENDFOLD
      ;FOLD F334 = AUS ;%{SE}%MKUKATPVW %CVW_SPS %VBOASG %P 2:F334 = AUS, 3: BOASG
         $FLAG[334] = FALSE
      ;ENDFOLD
      ;FOLD -- Quitt. Fraesen SK3 -- ;%{SE}%MKUKATPVW %CVW_COM %VCOMMENT %P 2:-- Quitt. Fraesen SK3 --, 3: VW_COMMENT
      ;ENDFOLD
      ;FOLD A1106 = (!F322 & !F830) + (F830 & A1106) + (E193 + A3505) & EIN ;%{SE}%MKUKATPVW %CVW_SPS %VBOASG %P 2:A1106 = (!F322 & !F830) + (F830 & A1106) + (E193 + A3505) & EIN, 3: BOASG
         $OUT[1106] = (NOT $FLAG[322] AND NOT $FLAG[830]) OR ($FLAG[830] AND $OUT[1106]) OR ($IN[193] OR $OUT[3505]) AND TRUE
      ;ENDFOLD
      ;FOLD A3936 = (!F174 & F175 & !F830) + (F830 & A3936) ;%{SE}%MKUKATPVW %CVW_SPS %VBOASG %P 2:A3936 = (!F174 & F175 & !F830) + (F830 & A3936), 3: BOASG
         $OUT[3936] = (NOT $FLAG[174] AND $FLAG[175] AND NOT $FLAG[830]) OR ($FLAG[830] AND $OUT[3936])
      ;ENDFOLD
      ;FOLD A3512 = (F174 & !F175 & !F830) + (F830 & A3512) ;%{SE}%MKUKATPVW %CVW_SPS %VBOASG %P 2:A3512 = (F174 & !F175 & !F830) + (F830 & A3512), 3: BOASG
         $OUT[3512] = ($FLAG[174] AND NOT $FLAG[175] AND NOT $FLAG[830]) OR ($FLAG[830] AND $OUT[3512])
      ;ENDFOLD
      ;FOLD SCHRITT 323 = A4039 & (!E1106 & !E1108 & !F830) ;%{SE}%MKUKATPVW %CVW_SPS %VST_CON %P 2:SCHRITT 323 = A4039 & (!E1106 & !E1108 & !F830), 3: ST_CON
         IF $OUT[4039] AND (NOT $IN[1106] AND NOT $IN[1108] AND NOT $FLAG[830]) THEN
            PREV_STEP[9] = APP_INT_STEP[9]
            APP_INT_STEP[9] = 323
         ENDIF
      ;ENDFOLD
   ;ENDFOLD
   ;FOLD SCHRITT 323 -- st. RZ3 # Ruecksetzen -- ;%{P}%MKUKATPVW,%CSTEP,%VST_NR,%P 1:SCHRITT, 2:323, 3: st. RZ3 # Ruecksetzen
      ;FOLD ;%{H}
         Case 323
      ;ENDFOLD
      ;FOLD -- Start Init Same AUS -- ;%{SE}%MKUKATPVW %CVW_COM %VCOMMENT %P 2:-- Start Init Same AUS --, 3: VW_COMMENT
      ;ENDFOLD
      ;FOLD A3514 = AUS ;%{SE}%MKUKATPVW %CVW_SPS %VBOASG %P 2:A3514 = AUS, 3: BOASG
         $OUT[3514] = FALSE
      ;ENDFOLD
      ;FOLD -- Start Spot AUS -- ;%{SE}%MKUKATPVW %CVW_COM %VCOMMENT %P 2:-- Start Spot AUS --, 3: VW_COMMENT
      ;ENDFOLD
      ;FOLD A3511 = AUS ;%{SE}%MKUKATPVW %CVW_SPS %VBOASG %P 2:A3511 = AUS, 3: BOASG
         $OUT[3511] = FALSE
      ;ENDFOLD
      ;FOLD -- Start Dress AUS -- ;%{SE}%MKUKATPVW %CVW_COM %VCOMMENT %P 2:-- Start Dress AUS --, 3: VW_COMMENT
      ;ENDFOLD
      ;FOLD A3510 = AUS ;%{SE}%MKUKATPVW %CVW_SPS %VBOASG %P 2:A3510 = AUS, 3: BOASG
         $OUT[3510] = FALSE
      ;ENDFOLD
      ;FOLD -- Start Init New AUS -- ;%{SE}%MKUKATPVW %CVW_COM %VCOMMENT %P 2:-- Start Init New AUS --, 3: VW_COMMENT
      ;ENDFOLD
      ;FOLD A3513 = AUS ;%{SE}%MKUKATPVW %CVW_SPS %VBOASG %P 2:A3513 = AUS, 3: BOASG
         $OUT[3513] = FALSE
      ;ENDFOLD
      ;FOLD -- Start Dress in Position AUS -- ;%{SE}%MKUKATPVW %CVW_COM %VCOMMENT %P 2:-- Start Dress in Position AUS --, 3: VW_COMMENT
      ;ENDFOLD
      ;FOLD A3935 = AUS ;%{SE}%MKUKATPVW %CVW_SPS %VBOASG %P 2:A3935 = AUS, 3: BOASG
         $OUT[3935] = FALSE
      ;ENDFOLD
      ;FOLD -- Start Dress Fin AUS -- ;%{SE}%MKUKATPVW %CVW_COM %VCOMMENT %P 2:-- Start Dress Fin AUS --, 3: VW_COMMENT
      ;ENDFOLD
      ;FOLD A3936 = AUS ;%{SE}%MKUKATPVW %CVW_SPS %VBOASG %P 2:A3936 = AUS, 3: BOASG
         $OUT[3936] = FALSE
      ;ENDFOLD
      ;FOLD -- Start StartAcknowledge AUS -- ;%{SE}%MKUKATPVW %CVW_COM %VCOMMENT %P 2:-- Start StartAcknowledge AUS --, 3: VW_COMMENT
      ;ENDFOLD
      ;FOLD A3512 = AUS ;%{SE}%MKUKATPVW %CVW_SPS %VBOASG %P 2:A3512 = AUS, 3: BOASG
         $OUT[3512] = FALSE
      ;ENDFOLD
      ;FOLD -- Ueberwachungszeit ServoGun SZ1 Messen -- ;%{SE}%MKUKATPVW %CVW_COM %VCOMMENT %P 2:-- Ueberwachungszeit ServoGun SZ1 Messen --, 3: VW_COMMENT
      ;ENDFOLD
      ;FOLD t9 ( EIN ) = -150[1/10Sek] ;%{SE}%MKUKATPVW %CVW_SPS %VTASG %P 2:t9 ( EIN ) = -150[1/10Sek], 3: TASG
         VW(#SET_TIME,TRUE,9,0,-150)
      ;ENDFOLD
      ;FOLD -- Fehler SK ruecksetzen -- ;%{SE}%MKUKATPVW %CVW_COM %VCOMMENT %P 2:-- Fehler SK ruecksetzen --, 3: VW_COMMENT
      ;ENDFOLD
      ;FOLD -- Fehler SK Messen AUS -- ;%{SE}%MKUKATPVW %CVW_COM %VCOMMENT %P 2:-- Fehler SK Messen AUS --, 3: VW_COMMENT
      ;ENDFOLD
      ;FOLD F326 = AUS ;%{SE}%MKUKATPVW %CVW_SPS %VBOASG %P 2:F326 = AUS, 3: BOASG
         $FLAG[326] = FALSE
      ;ENDFOLD
      ;FOLD SCHRITT 324 = A4039 & A3506 & A3505 & A3926 & !E1158 ;%{SE}%MKUKATPVW %CVW_SPS %VST_CON %P 2:SCHRITT 324 = A4039 & A3506 & A3505 & A3926 & !E1158, 3: ST_CON
         IF $OUT[4039] AND $OUT[3506] AND $OUT[3505] AND $OUT[3926] AND NOT $IN[1158] THEN
            PREV_STEP[9] = APP_INT_STEP[9]
            APP_INT_STEP[9] = 324
         ENDIF
      ;ENDFOLD
   ;ENDFOLD
   ;FOLD SCHRITT 324 -- st. RZ3 # Init Same -- ;%{P}%MKUKATPVW,%CSTEP,%VST_NR,%P 1:SCHRITT, 2:324, 3: st. RZ3 # Init Same
      ;FOLD ;%{H}
         Case 324
      ;ENDFOLD
      ;FOLD -- Kommentar -- ;%{SE}%MKUKATPVW %CVW_COM %VCOMMENT %P 2:-- Kommentar --, 3: VW_COMMENT
      ;ENDFOLD
      ;FOLD -- Messen nach Fraesen -- ;%{SE}%MKUKATPVW %CVW_COM %VCOMMENT %P 2:-- Messen nach Fraesen --, 3: VW_COMMENT
      ;ENDFOLD
      ;FOLD A3514 = EIN ;%{SE}%MKUKATPVW %CVW_SPS %VBOASG %P 2:A3514 = EIN, 3: BOASG
         $OUT[3514] = TRUE
      ;ENDFOLD
      ;FOLD A3510 = EIN ;%{SE}%MKUKATPVW %CVW_SPS %VBOASG %P 2:A3510 = EIN, 3: BOASG
         $OUT[3510] = TRUE
      ;ENDFOLD
      ;FOLD SCHRITT 325 = A4039 ;%{SE}%MKUKATPVW %CVW_SPS %VST_CON %P 2:SCHRITT 325 = A4039, 3: ST_CON
         IF $OUT[4039] THEN
            PREV_STEP[9] = APP_INT_STEP[9]
            APP_INT_STEP[9] = 325
         ENDIF
      ;ENDFOLD
   ;ENDFOLD
   ;FOLD SCHRITT 325 -- st. RZ3 # Auswertung -- ;%{P}%MKUKATPVW,%CSTEP,%VST_NR,%P 1:SCHRITT, 2:325, 3: st. RZ3 # Auswertung
      ;FOLD ;%{H}
         Case 325
      ;ENDFOLD
      ;FOLD -- Auswertung Messung -- ;%{SE}%MKUKATPVW %CVW_COM %VCOMMENT %P 2:-- Auswertung Messung --, 3: VW_COMMENT
      ;ENDFOLD
      ;FOLD SCHRITT 327 = A4039 & A3508 ;%{SE}%MKUKATPVW %CVW_SPS %VST_CON %P 2:SCHRITT 327 = A4039 & A3508, 3: ST_CON
         IF $OUT[4039] AND $OUT[3508] THEN
            PREV_STEP[9] = APP_INT_STEP[9]
            APP_INT_STEP[9] = 327
         ENDIF
      ;ENDFOLD
      ;FOLD SCHRITT 326 = A4039 & A3509 ;%{SE}%MKUKATPVW %CVW_SPS %VST_CON %P 2:SCHRITT 326 = A4039 & A3509, 3: ST_CON
         IF $OUT[4039] AND $OUT[3509] THEN
            PREV_STEP[9] = APP_INT_STEP[9]
            APP_INT_STEP[9] = 326
         ENDIF
      ;ENDFOLD
   ;ENDFOLD
   ;FOLD SCHRITT 326 -- st. RZ3 # Fehlerfall -- ;%{P}%MKUKATPVW,%CSTEP,%VST_NR,%P 1:SCHRITT, 2:326, 3: st. RZ3 # Fehlerfall
      ;FOLD ;%{H}
         Case 326
      ;ENDFOLD
      ;FOLD -- Start Init Same AUS -- ;%{SE}%MKUKATPVW %CVW_COM %VCOMMENT %P 2:-- Start Init Same AUS --, 3: VW_COMMENT
      ;ENDFOLD
      ;FOLD A3514 = AUS ;%{SE}%MKUKATPVW %CVW_SPS %VBOASG %P 2:A3514 = AUS, 3: BOASG
         $OUT[3514] = FALSE
      ;ENDFOLD
      ;FOLD -- Start Spot AUS -- ;%{SE}%MKUKATPVW %CVW_COM %VCOMMENT %P 2:-- Start Spot AUS --, 3: VW_COMMENT
      ;ENDFOLD
      ;FOLD A3511 = AUS ;%{SE}%MKUKATPVW %CVW_SPS %VBOASG %P 2:A3511 = AUS, 3: BOASG
         $OUT[3511] = FALSE
      ;ENDFOLD
      ;FOLD -- Start Dress AUS -- ;%{SE}%MKUKATPVW %CVW_COM %VCOMMENT %P 2:-- Start Dress AUS --, 3: VW_COMMENT
      ;ENDFOLD
      ;FOLD A3510 = AUS ;%{SE}%MKUKATPVW %CVW_SPS %VBOASG %P 2:A3510 = AUS, 3: BOASG
         $OUT[3510] = FALSE
      ;ENDFOLD
      ;FOLD -- Start Init New AUS -- ;%{SE}%MKUKATPVW %CVW_COM %VCOMMENT %P 2:-- Start Init New AUS --, 3: VW_COMMENT
      ;ENDFOLD
      ;FOLD A3513 = AUS ;%{SE}%MKUKATPVW %CVW_SPS %VBOASG %P 2:A3513 = AUS, 3: BOASG
         $OUT[3513] = FALSE
      ;ENDFOLD
      ;FOLD -- Start Dress in Position AUS -- ;%{SE}%MKUKATPVW %CVW_COM %VCOMMENT %P 2:-- Start Dress in Position AUS --, 3: VW_COMMENT
      ;ENDFOLD
      ;FOLD A3935 = AUS ;%{SE}%MKUKATPVW %CVW_SPS %VBOASG %P 2:A3935 = AUS, 3: BOASG
         $OUT[3935] = FALSE
      ;ENDFOLD
      ;FOLD -- Start Dress Fin AUS -- ;%{SE}%MKUKATPVW %CVW_COM %VCOMMENT %P 2:-- Start Dress Fin AUS --, 3: VW_COMMENT
      ;ENDFOLD
      ;FOLD A3936 = AUS ;%{SE}%MKUKATPVW %CVW_SPS %VBOASG %P 2:A3936 = AUS, 3: BOASG
         $OUT[3936] = FALSE
      ;ENDFOLD
      ;FOLD -- Start StartAcknowledge AUS -- ;%{SE}%MKUKATPVW %CVW_COM %VCOMMENT %P 2:-- Start StartAcknowledge AUS --, 3: VW_COMMENT
      ;ENDFOLD
      ;FOLD A3512 = AUS ;%{SE}%MKUKATPVW %CVW_SPS %VBOASG %P 2:A3512 = AUS, 3: BOASG
         $OUT[3512] = FALSE
      ;ENDFOLD
      ;FOLD -- Kommentar -- ;%{SE}%MKUKATPVW %CVW_COM %VCOMMENT %P 2:-- Kommentar --, 3: VW_COMMENT
      ;ENDFOLD
      ;FOLD -- RSK Sammelstoerung -- ;%{SE}%MKUKATPVW %CVW_COM %VCOMMENT %P 2:-- RSK Sammelstoerung --, 3: VW_COMMENT
      ;ENDFOLD
      ;FOLD F326 = EIN ;%{SE}%MKUKATPVW %CVW_SPS %VBOASG %P 2:F326 = EIN, 3: BOASG
         $FLAG[326] = TRUE
      ;ENDFOLD
      ;FOLD F329 = F326 ;%{SE}%MKUKATPVW %CVW_SPS %VBOASG %P 2:F329 = F326, 3: BOASG
         $FLAG[329] = $FLAG[326]
      ;ENDFOLD
      ;FOLD -- Flagbildung Wiederholfraesen -- ;%{SE}%MKUKATPVW %CVW_COM %VCOMMENT %P 2:-- Flagbildung Wiederholfraesen --, 3: VW_COMMENT
      ;ENDFOLD
      ;FOLD F749 = (F322 + F323 + F325 + F326 + F327 + F329) & !F748 ;%{SE}%MKUKATPVW %CVW_SPS %VBOASG %P 2:F749 = (F322 + F323 + F325 + F326 + F327 + F329) & !F748, 3: BOASG
         $FLAG[749] = ($FLAG[322] OR $FLAG[323] OR $FLAG[325] OR $FLAG[326] OR $FLAG[327] OR $FLAG[329]) AND NOT $FLAG[748]
      ;ENDFOLD
      ;FOLD SCHRITT 323 = A4039 & F326 & F329 & A3926 & (E26 + E27) ;%{SE}%MKUKATPVW %CVW_SPS %VST_CON %P 2:SCHRITT 323 = A4039 & F326 & F329 & A3926 & (E26 + E27), 3: ST_CON
         IF $OUT[4039] AND $FLAG[326] AND $FLAG[329] AND $OUT[3926] AND ($IN[26] OR $IN[27]) THEN
            PREV_STEP[9] = APP_INT_STEP[9]
            APP_INT_STEP[9] = 323
         ENDIF
      ;ENDFOLD
      ;FOLD SCHRITT 350 = A4039 & F326 & F329 & A3926 & A204 ;%{SE}%MKUKATPVW %CVW_SPS %VST_CON %P 2:SCHRITT 350 = A4039 & F326 & F329 & A3926 & A204, 3: ST_CON
         IF $OUT[4039] AND $FLAG[326] AND $FLAG[329] AND $OUT[3926] AND $OUT[204] THEN
            PREV_STEP[9] = APP_INT_STEP[9]
            APP_INT_STEP[9] = 350
         ENDIF
      ;ENDFOLD
   ;ENDFOLD
   ;FOLD SCHRITT 327 -- st. RZ3 # Acknowledge -- ;%{P}%MKUKATPVW,%CSTEP,%VST_NR,%P 1:SCHRITT, 2:327, 3: st. RZ3 # Acknowledge
      ;FOLD ;%{H}
         Case 327
      ;ENDFOLD
      ;FOLD -- ServoGun - StartAcknowledge -- ;%{SE}%MKUKATPVW %CVW_COM %VCOMMENT %P 2:-- ServoGun - StartAcknowledge --, 3: VW_COMMENT
      ;ENDFOLD
      ;FOLD -- Start Dress AUS -- ;%{SE}%MKUKATPVW %CVW_COM %VCOMMENT %P 2:-- Start Dress AUS --, 3: VW_COMMENT
      ;ENDFOLD
      ;FOLD A3510 = AUS ;%{SE}%MKUKATPVW %CVW_SPS %VBOASG %P 2:A3510 = AUS, 3: BOASG
         $OUT[3510] = FALSE
      ;ENDFOLD
      ;FOLD -- Start Init Same AUS -- ;%{SE}%MKUKATPVW %CVW_COM %VCOMMENT %P 2:-- Start Init Same AUS --, 3: VW_COMMENT
      ;ENDFOLD
      ;FOLD A3514 = AUS ;%{SE}%MKUKATPVW %CVW_SPS %VBOASG %P 2:A3514 = AUS, 3: BOASG
         $OUT[3514] = FALSE
      ;ENDFOLD
      ;FOLD -- Start StartAcknowledge EIN -- ;%{SE}%MKUKATPVW %CVW_COM %VCOMMENT %P 2:-- Start StartAcknowledge EIN --, 3: VW_COMMENT
      ;ENDFOLD
      ;FOLD A3512 = EIN ;%{SE}%MKUKATPVW %CVW_SPS %VBOASG %P 2:A3512 = EIN, 3: BOASG
         $OUT[3512] = TRUE
      ;ENDFOLD
      ;FOLD SCHRITT 329 = !F335 & A4039 & !A3507 ;%{SE}%MKUKATPVW %CVW_SPS %VST_CON %P 2:SCHRITT 329 = !F335 & A4039 & !A3507, 3: ST_CON
         IF NOT $FLAG[335] AND $OUT[4039] AND NOT $OUT[3507] THEN
            PREV_STEP[9] = APP_INT_STEP[9]
            APP_INT_STEP[9] = 329
         ENDIF
      ;ENDFOLD
      ;FOLD SCHRITT 329 = F335 & !F174 & A4039 & !A3507 ;%{SE}%MKUKATPVW %CVW_SPS %VST_CON %P 2:SCHRITT 329 = F335 & !F174 & A4039 & !A3507, 3: ST_CON
         IF $FLAG[335] AND NOT $FLAG[174] AND $OUT[4039] AND NOT $OUT[3507] THEN
            PREV_STEP[9] = APP_INT_STEP[9]
            APP_INT_STEP[9] = 329
         ENDIF
      ;ENDFOLD
      ;FOLD Schritt 390 = F335 & F174 & A4039 & !A3507 ;%{SE}%MKUKATPVW %CVW_SPS %VST_CON %P 2:Schritt 390 = F335 & F174 & A4039 & !A3507, 3: ST_CON
         IF $FLAG[335] AND $FLAG[174] AND $OUT[4039] AND NOT $OUT[3507] THEN
            PREV_STEP[9] = APP_INT_STEP[9]
            APP_INT_STEP[9] = 390
         ENDIF
      ;ENDFOLD
   ;ENDFOLD
   ;FOLD SCHRITT 329 -- st. RZ3 # Ruecksetzen -- ;%{P}%MKUKATPVW,%CSTEP,%VST_NR,%P 1:SCHRITT, 2:329, 3: st. RZ3 # Ruecksetzen
      ;FOLD ;%{H}
         Case 329
      ;ENDFOLD
      ;FOLD -- Start Init Same AUS -- ;%{SE}%MKUKATPVW %CVW_COM %VCOMMENT %P 2:-- Start Init Same AUS --, 3: VW_COMMENT
      ;ENDFOLD
      ;FOLD A3514 = AUS ;%{SE}%MKUKATPVW %CVW_SPS %VBOASG %P 2:A3514 = AUS, 3: BOASG
         $OUT[3514] = FALSE
      ;ENDFOLD
      ;FOLD -- Start Spot AUS -- ;%{SE}%MKUKATPVW %CVW_COM %VCOMMENT %P 2:-- Start Spot AUS --, 3: VW_COMMENT
      ;ENDFOLD
      ;FOLD A3511 = AUS ;%{SE}%MKUKATPVW %CVW_SPS %VBOASG %P 2:A3511 = AUS, 3: BOASG
         $OUT[3511] = FALSE
      ;ENDFOLD
      ;FOLD -- Start Dress AUS -- ;%{SE}%MKUKATPVW %CVW_COM %VCOMMENT %P 2:-- Start Dress AUS --, 3: VW_COMMENT
      ;ENDFOLD
      ;FOLD A3510 = AUS ;%{SE}%MKUKATPVW %CVW_SPS %VBOASG %P 2:A3510 = AUS, 3: BOASG
         $OUT[3510] = FALSE
      ;ENDFOLD
      ;FOLD -- Start Init New AUS -- ;%{SE}%MKUKATPVW %CVW_COM %VCOMMENT %P 2:-- Start Init New AUS --, 3: VW_COMMENT
      ;ENDFOLD
      ;FOLD A3513 = AUS ;%{SE}%MKUKATPVW %CVW_SPS %VBOASG %P 2:A3513 = AUS, 3: BOASG
         $OUT[3513] = FALSE
      ;ENDFOLD
      ;FOLD -- Start Dress in Position AUS -- ;%{SE}%MKUKATPVW %CVW_COM %VCOMMENT %P 2:-- Start Dress in Position AUS --, 3: VW_COMMENT
      ;ENDFOLD
      ;FOLD A3935 = AUS ;%{SE}%MKUKATPVW %CVW_SPS %VBOASG %P 2:A3935 = AUS, 3: BOASG
         $OUT[3935] = FALSE
      ;ENDFOLD
      ;FOLD -- Start Dress Fin AUS -- ;%{SE}%MKUKATPVW %CVW_COM %VCOMMENT %P 2:-- Start Dress Fin AUS --, 3: VW_COMMENT
      ;ENDFOLD
      ;FOLD A3936 = AUS ;%{SE}%MKUKATPVW %CVW_SPS %VBOASG %P 2:A3936 = AUS, 3: BOASG
         $OUT[3936] = FALSE
      ;ENDFOLD
      ;FOLD -- Start StartAcknowledge AUS -- ;%{SE}%MKUKATPVW %CVW_COM %VCOMMENT %P 2:-- Start StartAcknowledge AUS --, 3: VW_COMMENT
      ;ENDFOLD
      ;FOLD A3512 = AUS ;%{SE}%MKUKATPVW %CVW_SPS %VBOASG %P 2:A3512 = AUS, 3: BOASG
         $OUT[3512] = FALSE
      ;ENDFOLD
      ;FOLD bin30 ( EIN ) = 0 ;%{SE}%MKUKATPVW %CVW_SPS %VARIASG %P 2:bin30 ( EIN ) = 0, 3: ARIASG
         VW(#BINOUT,TRUE,30,0)
      ;ENDFOLD
      ;FOLD -- Fehler SK ruecksetzen -- ;%{SE}%MKUKATPVW %CVW_COM %VCOMMENT %P 2:-- Fehler SK ruecksetzen --, 3: VW_COMMENT
      ;ENDFOLD
      ;FOLD -- Druckvorgabe SK1/ServoGun -- ;%{SE}%MKUKATPVW %CVW_COM %VCOMMENT %P 2:-- Druckvorgabe SK1/ServoGun --, 3: VW_COMMENT
      ;ENDFOLD
      ;FOLD bin7 ( F174 ) = 41 ;%{SE}%MKUKATPVW %CVW_SPS %VARIASG %P 2:bin7 ( F174 ) = 41, 3: ARIASG
         VW(#BINOUT,$FLAG[174],7,41)
      ;ENDFOLD
      ;FOLD bin7 ( F175 ) = 51 ;%{SE}%MKUKATPVW %CVW_SPS %VARIASG %P 2:bin7 ( F175 ) = 51, 3: ARIASG
         VW(#BINOUT,$FLAG[175],7,51)
      ;ENDFOLD
      ;FOLD bin31 ( F174 ) = 41 ;%{SE}%MKUKATPVW %CVW_SPS %VARIASG %P 2:bin31 ( F174 ) = 41, 3: ARIASG
         VW(#BINOUT,$FLAG[174],31,41)
      ;ENDFOLD
      ;FOLD bin31 ( F175 ) = 51 ;%{SE}%MKUKATPVW %CVW_SPS %VARIASG %P 2:bin31 ( F175 ) = 51, 3: ARIASG
         VW(#BINOUT,$FLAG[175],31,51)
      ;ENDFOLD
      ;FOLD -- Wartezeit Programmwechsel SK -- ;%{SE}%MKUKATPVW %CVW_COM %VCOMMENT %P 2:-- Wartezeit Programmwechsel SK --, 3: VW_COMMENT
      ;ENDFOLD
      ;FOLD T8 ( !F334 ) = -2[1/10Sek] ;%{SE}%MKUKATPVW %CVW_SPS %VTASG %P 2:T8 ( !F334 ) = -2[1/10Sek], 3: TASG
         VW(#SET_TIME,NOT $FLAG[334],8,0,-2)
      ;ENDFOLD
      ;FOLD -- Hilfsflag SK Programmwechsel -- ;%{SE}%MKUKATPVW %CVW_COM %VCOMMENT %P 2:-- Hilfsflag SK Programmwechsel --, 3: VW_COMMENT
      ;ENDFOLD
      ;FOLD F334 = EIN ;%{SE}%MKUKATPVW %CVW_SPS %VBOASG %P 2:F334 = EIN, 3: BOASG
         $FLAG[334] = TRUE
      ;ENDFOLD
      ;FOLD t9 ( EIN ) = STOP ;%{SE}%MKUKATPVW %CVW_SPS %VTSTOP %P 2:t9 ( EIN ) = STOP, 3: TSTOP
         VW(#SET_TIME,TRUE,9,1,0)
      ;ENDFOLD
      ;FOLD SCHRITT 330 = T8 & A4039 & A3506 & A3505 & A3926 & !E1158 ;%{SE}%MKUKATPVW %CVW_SPS %VST_CON %P 2:SCHRITT 330 = T8 & A4039 & A3506 & A3505 & A3926 & !E1158, 3: ST_CON
         IF $TIMER_FLAG[8] AND $OUT[4039] AND $OUT[3506] AND $OUT[3505] AND $OUT[3926] AND NOT $IN[1158] THEN
            PREV_STEP[9] = APP_INT_STEP[9]
            APP_INT_STEP[9] = 330
         ENDIF
      ;ENDFOLD
   ;ENDFOLD
   ;FOLD SCHRITT 330 -- st. RZ3 # StartSpot -- ;%{P}%MKUKATPVW,%CSTEP,%VST_NR,%P 1:SCHRITT, 2:330, 3: st. RZ3 # StartSpot
      ;FOLD ;%{H}
         Case 330
      ;ENDFOLD
      ;FOLD -- Hilfsflag SK Programmwechsel -- ;%{SE}%MKUKATPVW %CVW_COM %VCOMMENT %P 2:-- Hilfsflag SK Programmwechsel --, 3: VW_COMMENT
      ;ENDFOLD
      ;FOLD F334 = AUS ;%{SE}%MKUKATPVW %CVW_SPS %VBOASG %P 2:F334 = AUS, 3: BOASG
         $FLAG[334] = FALSE
      ;ENDFOLD
      ;FOLD A3518 = A3519 & F731 ;%{SE}%MKUKATPVW %CVW_SPS %VBOASG %P 2:A3518 = A3519 & F731, 3: BOASG
         $OUT[3518] = $OUT[3519] AND $FLAG[731]
      ;ENDFOLD
      ;FOLD F748 = A3518 ;%{SE}%MKUKATPVW %CVW_SPS %VBOASG %P 2:F748 = A3518, 3: BOASG
         $FLAG[748] = $OUT[3518]
      ;ENDFOLD
      ;FOLD -- ServoGun - Start Spot EIN -- ;%{SE}%MKUKATPVW %CVW_COM %VCOMMENT %P 2:-- ServoGun - Start Spot EIN --, 3: VW_COMMENT
      ;ENDFOLD
      ;FOLD A3511 = EIN ;%{SE}%MKUKATPVW %CVW_SPS %VBOASG %P 2:A3511 = EIN, 3: BOASG
         $OUT[3511] = TRUE
      ;ENDFOLD
      ;FOLD F749 = AUS ;%{SE}%MKUKATPVW %CVW_SPS %VBOASG %P 2:F749 = AUS, 3: BOASG
         $FLAG[749] = FALSE
      ;ENDFOLD
      ;FOLD SCHRITT 331 = A4039 ;%{SE}%MKUKATPVW %CVW_SPS %VST_CON %P 2:SCHRITT 331 = A4039, 3: ST_CON
         IF $OUT[4039] THEN
            PREV_STEP[9] = APP_INT_STEP[9]
            APP_INT_STEP[9] = 331
         ENDIF
      ;ENDFOLD
   ;ENDFOLD
   ;FOLD SCHRITT 331 -- st. RZ3 # Auswertung -- ;%{P}%MKUKATPVW,%CSTEP,%VST_NR,%P 1:SCHRITT, 2:331, 3: st. RZ3 # Auswertung
      ;FOLD ;%{H}
         Case 331
      ;ENDFOLD
      ;FOLD -- Auswertung -- ;%{SE}%MKUKATPVW %CVW_COM %VCOMMENT %P 2:-- Auswertung --, 3: VW_COMMENT
      ;ENDFOLD
      ;FOLD Schritt 332 = A3509 ;%{SE}%MKUKATPVW %CVW_SPS %VST_CON %P 2:Schritt 332 = A3509, 3: ST_CON
         IF $OUT[3509] THEN
            PREV_STEP[9] = APP_INT_STEP[9]
            APP_INT_STEP[9] = 332
         ENDIF
      ;ENDFOLD
      ;FOLD SCHRITT 333 = A3508 & E1024 & !E1026 ;%{SE}%MKUKATPVW %CVW_SPS %VST_CON %P 2:SCHRITT 333 = A3508 & E1024 & !E1026, 3: ST_CON
         IF $OUT[3508] AND $IN[1024] AND NOT $IN[1026] THEN
            PREV_STEP[9] = APP_INT_STEP[9]
            APP_INT_STEP[9] = 333
         ENDIF
      ;ENDFOLD
   ;ENDFOLD
   ;FOLD SCHRITT 332 -- st. RZ3 # Fehler Schweissung -- ;%{P}%MKUKATPVW,%CSTEP,%VST_NR,%P 1:SCHRITT, 2:332, 3: st. RZ3 # Fehler Schweissung
      ;FOLD ;%{H}
         Case 332
      ;ENDFOLD
      ;FOLD -- Start Init Same AUS -- ;%{SE}%MKUKATPVW %CVW_COM %VCOMMENT %P 2:-- Start Init Same AUS --, 3: VW_COMMENT
      ;ENDFOLD
      ;FOLD A3514 = AUS ;%{SE}%MKUKATPVW %CVW_SPS %VBOASG %P 2:A3514 = AUS, 3: BOASG
         $OUT[3514] = FALSE
      ;ENDFOLD
      ;FOLD -- Start Spot AUS -- ;%{SE}%MKUKATPVW %CVW_COM %VCOMMENT %P 2:-- Start Spot AUS --, 3: VW_COMMENT
      ;ENDFOLD
      ;FOLD A3511 = AUS ;%{SE}%MKUKATPVW %CVW_SPS %VBOASG %P 2:A3511 = AUS, 3: BOASG
         $OUT[3511] = FALSE
      ;ENDFOLD
      ;FOLD -- Start Dress AUS -- ;%{SE}%MKUKATPVW %CVW_COM %VCOMMENT %P 2:-- Start Dress AUS --, 3: VW_COMMENT
      ;ENDFOLD
      ;FOLD A3510 = AUS ;%{SE}%MKUKATPVW %CVW_SPS %VBOASG %P 2:A3510 = AUS, 3: BOASG
         $OUT[3510] = FALSE
      ;ENDFOLD
      ;FOLD -- Start Init New AUS -- ;%{SE}%MKUKATPVW %CVW_COM %VCOMMENT %P 2:-- Start Init New AUS --, 3: VW_COMMENT
      ;ENDFOLD
      ;FOLD A3513 = AUS ;%{SE}%MKUKATPVW %CVW_SPS %VBOASG %P 2:A3513 = AUS, 3: BOASG
         $OUT[3513] = FALSE
      ;ENDFOLD
      ;FOLD -- Start Dress in Position AUS -- ;%{SE}%MKUKATPVW %CVW_COM %VCOMMENT %P 2:-- Start Dress in Position AUS --, 3: VW_COMMENT
      ;ENDFOLD
      ;FOLD A3935 = AUS ;%{SE}%MKUKATPVW %CVW_SPS %VBOASG %P 2:A3935 = AUS, 3: BOASG
         $OUT[3935] = FALSE
      ;ENDFOLD
      ;FOLD -- Start Dress Fin AUS -- ;%{SE}%MKUKATPVW %CVW_COM %VCOMMENT %P 2:-- Start Dress Fin AUS --, 3: VW_COMMENT
      ;ENDFOLD
      ;FOLD A3936 = AUS ;%{SE}%MKUKATPVW %CVW_SPS %VBOASG %P 2:A3936 = AUS, 3: BOASG
         $OUT[3936] = FALSE
      ;ENDFOLD
